KUKA KRL program: EPS_2_251692_SAMH04_A_20251205090700.src

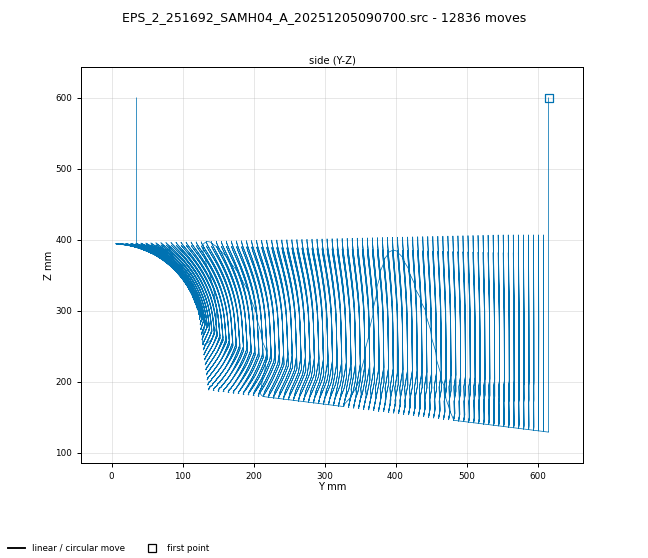
[picture p0: tool path of EPS_2_251692_SAMH04_A_20251205090700.src, 12836 of 12838 moves have a stored position in this frame; points joined in program order, loops and branches not executed]
&ACCESS RVP
&REL 4
&COMMENT QRS 19112012
&PARAM EDITMASK = *
DEF PART()
EXT BAS (BAS_COMMAND :IN,REAL :IN )
INT I
BAS (#INITMOV,0 )

;KUKA QRS Post kuka4.cps  Date:22-06-2017 !

File_ID=2946

QRS_PRE_INIT()

;Init var - Until changes are made in qrs_pre_init
Outlet_Square_prg=0
Inlet_1_Square_prg=0
Inlet_2_Square_prg=0
Inlet_3_Square_prg=0
Inlet_4_Square_prg=0
Inlet_5_Square_prg=0

Outlet_1={X 0.000, Y 546.330, Z 306.500, B 0.000, E1 0.000 }
Inlet_1={X 0.000, Y 548.110, Z 281.500, B 0.000, E1 180.000 }
Outlet_1_type=201
Inlet_1_type=201
;QRS#1=Sidecore dimensions
;QRS#2=200-8" PVC SDR 35
;QRS#3=200-8" PVC SDR 35
;QRS#4=
;QRS#5=
;QRS#6=
;QRS#7=
;QRS#8=
;QRS#9=12-08 PSX
;QRS#10=12-08 PSX
;QRS#11=
;QRS#12=
;QRS#13=
;QRS#14=
;QRS#15=
;QRS#16=1220x127x686 2,25'
;QRS#17=EPS Height
;QRS#18=407
;QRS#19=*
;QRS#20= UPDATED VERSION 22-06-2017
;QRS#21=*
Outlet_Square=0100
Inlet_1_Square=0100
Inlet_2_Square=0
Inlet_3_Square=0
Inlet_4_Square=0
Inlet_5_Square=0
Mill_Square=1
Outlet_Square_Prg=204
Inlet_1_Square_prg=204

QRS_INIT()

$ADVANCE=5

; T1
PTP {E1 173.62,E2 173.62}
PTP {X 0,Y 615.48,A -85,B 0,C 180,E1 173.62,E2 173.62,E3 0,E4 0,E5 0,E6 0}
QRS_SPEED_INIT()
LIN {X 0,Y 615.48,Z 600,A -85,B 0,C 180,E1 173.62,E2 173.62,E3 0,E4 0,E5 0,E6 0} C_VEL
LIN {X 0,Y 615.48,Z 139.368,A -85,B 0,C 180,E1 173.62,E2 173.62} C_VEL
LIN {X 0,Y 615.48,Z 131.192,A -85,B 0,C 180,E1 173.62,E2 173.62} C_VEL
LIN {X 0,Y 615.471,Z 129.192,A -85,B 0,C 180,E1 173.434,E2 173.434} C_VEL
LIN {X 0,Y 615.484,Z 129.195,A -85,B 0,C 180,E1 170.801,E2 170.801} C_VEL
LIN {X 0,Y 615.485,Z 129.184,A -85,B 0,C 180,E1 168.139,E2 168.139} C_VEL
LIN {X 0,Y 615.481,Z 129.196,A -85,B 0,C 180,E1 165.451,E2 165.451} C_VEL
LIN {X 0,Y 615.483,Z 129.188,A -85,B 0,C 180,E1 162.729,E2 162.729} C_VEL
LIN {X 0,Y 615.475,Z 129.189,A -85,B 0,C 180,E1 159.967,E2 159.967} C_VEL
LIN {X 0,Y 615.483,Z 129.194,A -85,B 0,C 180,E1 157.155,E2 157.155} C_VEL
LIN {X 0,Y 615.481,Z 129.186,A -85,B 0,C 180,E1 154.284,E2 154.284} C_VEL
LIN {X 0,Y 615.494,Z 129.199,A -85,B 0,C 180,E1 151.548,E2 151.548} C_VEL
LIN {X 0,Y 615.485,Z 129.185,A -85,B 0,C 180,E1 148.914,E2 148.914} C_VEL
LIN {X 0,Y 615.483,Z 129.186,A -85,B 0,C 180,E1 146.466,E2 146.466} C_VEL
LIN {X 0,Y 615.481,Z 129.195,A -85,B 0,C 180,E1 143.575,E2 143.575} C_VEL
LIN {X 0,Y 615.494,Z 129.181,A -85,B 0,C 180,E1 140.937,E2 140.937} C_VEL
LIN {X 0,Y 615.488,Z 129.199,A -85,B 0,C 180,E1 137.92,E2 137.92} C_VEL
LIN {X 0,Y 615.495,Z 129.182,A -85,B 0,C 180,E1 134.932,E2 134.932} C_VEL
LIN {X 0,Y 615.489,Z 129.198,A -85,B 0,C 180,E1 132.08,E2 132.08} C_VEL
LIN {X 0,Y 615.47,Z 129.192,A -85,B 0,C 180,E1 129.751,E2 129.751} C_VEL
LIN {X 0,Y 615.488,Z 129.186,A -85,B 0,C 180,E1 126.936,E2 126.936} C_VEL
LIN {X 0,Y 615.47,Z 129.194,A -85,B 0,C 180,E1 124.023,E2 124.023} C_VEL
LIN {X 0,Y 615.469,Z 129.188,A -85,B 0,C 180,E1 121.686,E2 121.686} C_VEL
LIN {X 0,Y 615.486,Z 129.184,A -85,B 0,C 180,E1 119.406,E2 119.406} C_VEL
LIN {X 0,Y 615.478,Z 129.197,A -85,B 0,C 180,E1 116.444,E2 116.444} C_VEL
LIN {X 0,Y 615.465,Z 129.189,A -85,B 0,C 180,E1 114.003,E2 114.003} C_VEL
LIN {X 0,Y 615.495,Z 129.184,A -85,B 0,C 180,E1 111.432,E2 111.432} C_VEL
LIN {X 0,Y 615.495,Z 129.385,A -85,B 0,C 180,E1 109.468,E2 109.468} C_VEL
LIN {X 0,Y 615.486,Z 146.128,A -85,B 0,C 180,E1 106.757,E2 106.757} C_VEL
LIN {X 0,Y 615.491,Z 164.181,A -85,B 0,C 180,E1 103.874,E2 103.874} C_VEL
LIN {X 0,Y 615.487,Z 170.814,A -85,B 0,C 180,E1 102.824,E2 102.824} C_VEL
LIN {X 0,Y 615.486,Z 278.794,A -85,B 0,C 180,E1 101.527,E2 101.527} C_VEL
LIN {X 0,Y 615.476,Z 291.742,A -85,B 0,C 180,E1 101.235,E2 101.235} C_VEL
LIN {X 0,Y 615.488,Z 303.661,A -85,B 0,C 180,E1 100.84,E2 100.84} C_VEL
LIN {X 0,Y 615.481,Z 316.197,A -85,B 0,C 180,E1 100.278,E2 100.278} C_VEL
LIN {X 0,Y 615.494,Z 327.576,A -85,B 0,C 180,E1 99.613,E2 99.613} C_VEL
LIN {X 0,Y 615.498,Z 337.823,A -85,B 0,C 180,E1 98.867,E2 98.867} C_VEL
LIN {X 0,Y 615.498,Z 347.034,A -85,B 0,C 180,E1 98.041,E2 98.041} C_VEL
LIN {X 0,Y 615.499,Z 355.892,A -85,B 0,C 180,E1 97.057,E2 97.057} C_VEL
LIN {X 0,Y 615.497,Z 363.123,A -85,B 0,C 180,E1 96.063,E2 96.063} C_VEL
LIN {X 0,Y 615.497,Z 367.958,A -85,B 0,C 180,E1 95.241,E2 95.241} C_VEL
LIN {X 0,Y 615.494,Z 372.658,A -85,B 0,C 180,E1 94.256,E2 94.256} C_VEL
LIN {X 0,Y 615.494,Z 376.254,A -85,B 0,C 180,E1 93.273,E2 93.273} C_VEL
LIN {X 0,Y 615.496,Z 378.115,A -85,B 0,C 180,E1 92.618,E2 92.618} C_VEL
LIN {X 0,Y 615.5,Z 379.533,A -85,B 0,C 180,E1 91.963,E2 91.963} C_VEL
LIN {X 0,Y 615.496,Z 381.141,A -85,B 0,C 180,E1 90.654,E2 90.654} C_VEL
LIN {X 0,Y 615.495,Z 381.384,A -85,B 0,C 180,E1 90,E2 90} C_VEL
LIN {X 0,Y 615.495,Z 381.206,A -85,B 0,C 180,E1 89.346,E2 89.346} C_VEL
LIN {X 0,Y 615.5,Z 379.682,A -85,B 0,C 180,E1 88.037,E2 88.037} C_VEL
LIN {X 0,Y 615.498,Z 378.341,A -85,B 0,C 180,E1 87.382,E2 87.382} C_VEL
LIN {X 0,Y 615.496,Z 375.494,A -85,B 0,C 180,E1 86.399,E2 86.399} C_VEL
LIN {X 0,Y 615.498,Z 371.634,A -85,B 0,C 180,E1 85.416,E2 85.416} C_VEL
LIN {X 0,Y 615.498,Z 366.652,A -85,B 0,C 180,E1 84.43,E2 84.43} C_VEL
LIN {X 0,Y 615.496,Z 360.208,A -85,B 0,C 180,E1 83.418,E2 83.418} C_VEL
LIN {X 0,Y 615.497,Z 352.537,A -85,B 0,C 180,E1 82.455,E2 82.455} C_VEL
LIN {X 0,Y 615.498,Z 342.759,A -85,B 0,C 180,E1 81.464,E2 81.464} C_VEL
LIN {X 0,Y 615.498,Z 332.494,A -85,B 0,C 180,E1 80.636,E2 80.636} C_VEL
LIN {X 0,Y 615.48,Z 320.933,A -85,B 0,C 180,E1 79.889,E2 79.889} C_VEL
LIN {X 0,Y 615.494,Z 309.074,A -85,B 0,C 180,E1 79.293,E2 79.293} C_VEL
LIN {X 0,Y 615.478,Z 296.164,A -85,B 0,C 180,E1 78.807,E2 78.807} C_VEL
LIN {X 0,Y 615.485,Z 283.563,A -85,B 0,C 180,E1 78.473,E2 78.473} C_VEL
LIN {X 0,Y 615.493,Z 270.44,A -85,B 0,C 180,E1 78.265,E2 78.265} C_VEL
LIN {X 0,Y 615.493,Z 170.852,A -85,B 0,C 180,E1 77.093,E2 77.093} C_VEL
LIN {X 0,Y 615.491,Z 152.002,A -85,B 0,C 180,E1 74.095,E2 74.095} C_VEL
LIN {X 0,Y 615.477,Z 134.992,A -85,B 0,C 180,E1 71.354,E2 71.354} C_VEL
LIN {X 0,Y 615.489,Z 129.185,A -85,B 0,C 180,E1 70.402,E2 70.402} C_VEL
LIN {X 0,Y 615.46,Z 129.193,A -85,B 0,C 180,E1 67.661,E2 67.661} C_VEL
LIN {X 0,Y 615.492,Z 129.195,A -85,B 0,C 180,E1 65.009,E2 65.009} C_VEL
LIN {X 0,Y 615.462,Z 129.19,A -85,B 0,C 180,E1 62.084,E2 62.084} C_VEL
LIN {X 0,Y 615.465,Z 129.194,A -85,B 0,C 180,E1 59.839,E2 59.839} C_VEL
LIN {X 0,Y 615.482,Z 129.2,A -85,B 0,C 180,E1 57.542,E2 57.542} C_VEL
LIN {X 0,Y 615.489,Z 129.192,A -85,B 0,C 180,E1 55.185,E2 55.185} C_VEL
LIN {X 0,Y 615.491,Z 129.183,A -85,B 0,C 180,E1 52.758,E2 52.758} C_VEL
LIN {X 0,Y 615.476,Z 129.197,A -85,B 0,C 180,E1 49.913,E2 49.913} C_VEL
LIN {X 0,Y 615.488,Z 129.184,A -85,B 0,C 180,E1 46.953,E2 46.953} C_VEL
LIN {X 0,Y 615.475,Z 129.195,A -85,B 0,C 180,E1 44.151,E2 44.151} C_VEL
LIN {X 0,Y 615.484,Z 129.19,A -85,B 0,C 180,E1 41.474,E2 41.474} C_VEL
LIN {X 0,Y 615.482,Z 129.184,A -85,B 0,C 180,E1 38.905,E2 38.905} C_VEL
LIN {X 0,Y 615.476,Z 129.194,A -85,B 0,C 180,E1 36.426,E2 36.426} C_VEL
LIN {X 0,Y 615.485,Z 129.186,A -85,B 0,C 180,E1 33.534,E2 33.534} C_VEL
LIN {X 0,Y 615.477,Z 129.188,A -85,B 0,C 180,E1 30.921,E2 30.921} C_VEL
LIN {X 0,Y 615.489,Z 129.198,A -85,B 0,C 180,E1 28.451,E2 28.451} C_VEL
LIN {X 0,Y 615.486,Z 129.184,A -85,B 0,C 180,E1 25.569,E2 25.569} C_VEL
LIN {X 0,Y 615.48,Z 129.193,A -85,B 0,C 180,E1 22.845,E2 22.845} C_VEL
LIN {X 0,Y 615.489,Z 129.202,A -85,B 0,C 180,E1 20.558,E2 20.558} C_VEL
LIN {X 0,Y 615.478,Z 129.187,A -85,B 0,C 180,E1 17.957,E2 17.957} C_VEL
LIN {X 0,Y 615.481,Z 129.189,A -85,B 0,C 180,E1 15.226,E2 15.226} C_VEL
LIN {X 0,Y 615.481,Z 129.195,A -85,B 0,C 180,E1 12.53,E2 12.53} C_VEL
LIN {X 0,Y 615.493,Z 129.182,A -85,B 0,C 180,E1 9.862,E2 9.862} C_VEL
LIN {X 0,Y 615.486,Z 129.195,A -85,B 0,C 180,E1 7.216,E2 7.216} C_VEL
LIN {X 0,Y 615.472,Z 129.192,A -85,B 0,C 180,E1 4.585,E2 4.585} C_VEL
LIN {X 0,Y 615.5,Z 129.181,A -85,B 0,C 180,E1 1.963,E2 1.963} C_VEL
LIN {X 0,Y 615.492,Z 129.197,A -85,B 0,C 180,E1 -0.654,E2 -0.654} C_VEL
LIN {X 0,Y 615.468,Z 129.191,A -85,B 0,C 180,E1 -3.273,E2 -3.273} C_VEL
LIN {X 0,Y 615.498,Z 129.182,A -85,B 0,C 180,E1 -5.898,E2 -5.898} C_VEL
LIN {X 0,Y 615.49,Z 129.202,A -85,B 0,C 180,E1 -8.537,E2 -8.537} C_VEL
LIN {X 0,Y 615.465,Z 129.19,A -85,B 0,C 180,E1 -11.194,E2 -11.194} C_VEL
LIN {X 0,Y 615.49,Z 129.188,A -85,B 0,C 180,E1 -13.935,E2 -13.935} C_VEL
LIN {X 0,Y 615.475,Z 129.196,A -85,B 0,C 180,E1 -16.587,E2 -16.587} C_VEL
LIN {X 0,Y 615.477,Z 129.186,A -85,B 0,C 180,E1 -19.338,E2 -19.338} C_VEL
LIN {X 0,Y 615.477,Z 129.198,A -85,B 0,C 180,E1 -22.344,E2 -22.344} C_VEL
LIN {X 0,Y 615.461,Z 129.189,A -85,B 0,C 180,E1 -24.993,E2 -24.993} C_VEL
LIN {X 0,Y 615.487,Z 129.201,A -85,B 0,C 180,E1 -27.915,E2 -27.915} C_VEL
LIN {X 0,Y 615.473,Z 129.197,A -85,B 0,C 180,E1 -30.161,E2 -30.161} C_VEL
LIN {X 0,Y 615.454,Z 129.193,A -85,B 0,C 180,E1 -32.46,E2 -32.46} C_VEL
LIN {X 0,Y 615.462,Z 129.189,A -85,B 0,C 180,E1 -34.817,E2 -34.817} C_VEL
LIN {X 0,Y 615.496,Z 129.187,A -85,B 0,C 180,E1 -37.242,E2 -37.242} C_VEL
LIN {X 0,Y 615.453,Z 129.196,A -85,B 0,C 180,E1 -40.085,E2 -40.085} C_VEL
LIN {X 0,Y 615.448,Z 129.192,A -85,B 0,C 180,E1 -42.357,E2 -42.357} C_VEL
LIN {X 0,Y 615.497,Z 129.189,A -85,B 0,C 180,E1 -45.068,E2 -45.068} C_VEL
LIN {X 0,Y 615.449,Z 129.195,A -85,B 0,C 180,E1 -47.924,E2 -47.924} C_VEL
LIN {X 0,Y 615.444,Z 129.193,A -85,B 0,C 180,E1 -50.247,E2 -50.247} C_VEL
LIN {X 0,Y 615.49,Z 129.197,A -85,B 0,C 180,E1 -53.063,E2 -53.063} C_VEL
LIN {X 0,Y 615.44,Z 129.194,A -85,B 0,C 180,E1 -55.975,E2 -55.975} C_VEL
LIN {X 0,Y 615.488,Z 129.199,A -85,B 0,C 180,E1 -58.914,E2 -58.914} C_VEL
LIN {X 0,Y 615.441,Z 129.196,A -85,B 0,C 180,E1 -61.558,E2 -61.558} C_VEL
LIN {X 0,Y 615.438,Z 129.196,A -85,B 0,C 180,E1 -63.554,E2 -63.554} C_VEL
LIN {X 0,Y 615.444,Z 129.194,A -85,B 0,C 180,E1 -66.001,E2 -66.001} C_VEL
LIN {X 0,Y 615.449,Z 129.225,A -85,B 0,C 180,E1 -68.039,E2 -68.039} C_VEL
LIN {X 0,Y 615.481,Z 149.073,A -85,B 0,C 180,E1 -70.835,E2 -70.835} C_VEL
LIN {X 0,Y 615.46,Z 167.661,A -85,B 0,C 180,E1 -73.413,E2 -73.413} C_VEL
LIN {X 0,Y 615.483,Z 187.465,A -85,B 0,C 180,E1 -76.126,E2 -76.126} C_VEL
LIN {X 0,Y 615.462,Z 195.117,A -85,B 0,C 180,E1 -77.134,E2 -77.134} C_VEL
LIN {X 0,Y 615.488,Z 302.834,A -85,B 0,C 180,E1 -78.411,E2 -78.411} C_VEL
LIN {X 0,Y 615.477,Z 315.348,A -85,B 0,C 180,E1 -78.682,E2 -78.682} C_VEL
LIN {X 0,Y 615.488,Z 328.617,A -85,B 0,C 180,E1 -79.113,E2 -79.113} C_VEL
LIN {X 0,Y 615.477,Z 340.48,A -85,B 0,C 180,E1 -79.639,E2 -79.639} C_VEL
LIN {X 0,Y 615.494,Z 351.995,A -85,B 0,C 180,E1 -80.304,E2 -80.304} C_VEL
LIN {X 0,Y 615.499,Z 362.342,A -85,B 0,C 180,E1 -81.05,E2 -81.05} C_VEL
LIN {X 0,Y 615.497,Z 370.812,A -85,B 0,C 180,E1 -81.794,E2 -81.794} C_VEL
LIN {X 0,Y 615.498,Z 378.607,A -85,B 0,C 180,E1 -82.62,E2 -82.62} C_VEL
LIN {X 0,Y 615.496,Z 386.203,A -85,B 0,C 180,E1 -83.608,E2 -83.608} C_VEL
LIN {X 0,Y 615.498,Z 393.205,A -85,B 0,C 180,E1 -84.759,E2 -84.759} C_VEL
LIN {X 0,Y 615.494,Z 397.852,A -85,B 0,C 180,E1 -85.744,E2 -85.744} C_VEL
LIN {X 0,Y 615.494,Z 401.399,A -85,B 0,C 180,E1 -86.727,E2 -86.727} C_VEL
LIN {X 0,Y 615.497,Z 403.233,A -85,B 0,C 180,E1 -87.382,E2 -87.382} C_VEL
LIN {X 0,Y 615.5,Z 404.607,A -85,B 0,C 180,E1 -88.037,E2 -88.037} C_VEL
LIN {X 0,Y 615.496,Z 406.173,A -85,B 0,C 180,E1 -89.346,E2 -89.346} C_VEL
LIN {X 0,Y 615.494,Z 406.389,A -85,B 0,C 180,E1 -90,E2 -90} C_VEL
LIN {X 0,Y 615.495,Z 405.58,A -85,B 0,C 180,E1 -91.309,E2 -91.309} C_VEL
LIN {X 0,Y 615.5,Z 404.607,A -85,B 0,C 180,E1 -91.963,E2 -91.963} C_VEL
LIN {X 0,Y 615.497,Z 403.233,A -85,B 0,C 180,E1 -92.618,E2 -92.618} C_VEL
LIN {X 0,Y 615.496,Z 400.349,A -85,B 0,C 180,E1 -93.601,E2 -93.601} C_VEL
LIN {X 0,Y 615.498,Z 396.441,A -85,B 0,C 180,E1 -94.584,E2 -94.584} C_VEL
LIN {X 0,Y 615.499,Z 391.405,A -85,B 0,C 180,E1 -95.57,E2 -95.57} C_VEL
LIN {X 0,Y 615.497,Z 384.869,A -85,B 0,C 180,E1 -96.583,E2 -96.583} C_VEL
LIN {X 0,Y 615.497,Z 377.133,A -85,B 0,C 180,E1 -97.545,E2 -97.545} C_VEL
LIN {X 0,Y 615.498,Z 369.045,A -85,B 0,C 180,E1 -98.371,E2 -98.371} C_VEL
LIN {X 0,Y 615.499,Z 359.167,A -85,B 0,C 180,E1 -99.199,E2 -99.199} C_VEL
LIN {X 0,Y 615.488,Z 347.982,A -85,B 0,C 180,E1 -99.945,E2 -99.945} C_VEL
LIN {X 0,Y 615.482,Z 337.023,A -85,B 0,C 180,E1 -100.527,E2 -100.527} C_VEL
LIN {X 0,Y 615.48,Z 324.49,A -85,B 0,C 180,E1 -101.04,E2 -101.04} C_VEL
LIN {X 0,Y 615.479,Z 312.067,A -85,B 0,C 180,E1 -101.402,E2 -101.402} C_VEL
LIN {X 0,Y 615.493,Z 298.465,A -85,B 0,C 180,E1 -101.652,E2 -101.652} C_VEL
LIN {X 0,Y 615.463,Z 194.734,A -85,B 0,C 180,E1 -102.887,E2 -102.887} C_VEL
LIN {X 0,Y 615.498,Z 173.851,A -85,B 0,C 180,E1 -105.735,E2 -105.735} C_VEL
LIN {X 0,Y 615.49,Z 153.088,A -85,B 0,C 180,E1 -108.605,E2 -108.605} C_VEL
LIN {X 0,Y 615.498,Z 132.948,A -85,B 0,C 180,E1 -111.431,E2 -111.431} C_VEL
LIN {X 0,Y 615.447,Z 129.194,A -85,B 0,C 180,E1 -111.983,E2 -111.983} C_VEL
LIN {X 0,Y 615.434,Z 129.195,A -85,B 0,C 180,E1 -114.274,E2 -114.274} C_VEL
LIN {X 0,Y 615.491,Z 129.2,A -85,B 0,C 180,E1 -117.045,E2 -117.045} C_VEL
LIN {X 0,Y 615.451,Z 129.192,A -85,B 0,C 180,E1 -119.788,E2 -119.788} C_VEL
LIN {X 0,Y 615.439,Z 129.197,A -85,B 0,C 180,E1 -122.323,E2 -122.323} C_VEL
LIN {X 0,Y 615.49,Z 129.2,A -85,B 0,C 180,E1 -124.815,E2 -124.815} C_VEL
LIN {X 0,Y 615.488,Z 129.189,A -85,B 0,C 180,E1 -127.242,E2 -127.242} C_VEL
LIN {X 0,Y 615.443,Z 129.193,A -85,B 0,C 180,E1 -129.753,E2 -129.753} C_VEL
LIN {X 0,Y 615.466,Z 129.198,A -85,B 0,C 180,E1 -132.355,E2 -132.355} C_VEL
LIN {X 0,Y 615.491,Z 129.187,A -85,B 0,C 180,E1 -135.068,E2 -135.068} C_VEL
LIN {X 0,Y 615.447,Z 129.193,A -85,B 0,C 180,E1 -137.643,E2 -137.643} C_VEL
LIN {X 0,Y 615.48,Z 129.199,A -85,B 0,C 180,E1 -140.249,E2 -140.249} C_VEL
LIN {X 0,Y 615.473,Z 129.188,A -85,B 0,C 180,E1 -143.065,E2 -143.065} C_VEL
LIN {X 0,Y 615.455,Z 129.19,A -85,B 0,C 180,E1 -145.304,E2 -145.304} C_VEL
LIN {X 0,Y 615.456,Z 129.195,A -85,B 0,C 180,E1 -147.674,E2 -147.674} C_VEL
LIN {X 0,Y 615.497,Z 129.198,A -85,B 0,C 180,E1 -150.204,E2 -150.204} C_VEL
LIN {X 0,Y 615.464,Z 129.188,A -85,B 0,C 180,E1 -152.959,E2 -152.959} C_VEL
LIN {X 0,Y 615.461,Z 129.189,A -85,B 0,C 180,E1 -155.007,E2 -155.007} C_VEL
LIN {X 0,Y 615.473,Z 129.198,A -85,B 0,C 180,E1 -157.657,E2 -157.657} C_VEL
LIN {X 0,Y 615.477,Z 129.186,A -85,B 0,C 180,E1 -160.662,E2 -160.662} C_VEL
LIN {X 0,Y 615.467,Z 129.197,A -85,B 0,C 180,E1 -163.413,E2 -163.413} C_VEL
LIN {X 0,Y 615.492,Z 129.187,A -85,B 0,C 180,E1 -166.126,E2 -166.126} C_VEL
LIN {X 0,Y 615.462,Z 129.19,A -85,B 0,C 180,E1 -168.806,E2 -168.806} C_VEL
LIN {X 0,Y 615.488,Z 129.202,A -85,B 0,C 180,E1 -171.463,E2 -171.463} C_VEL
LIN {X 0,Y 615.498,Z 129.182,A -85,B 0,C 180,E1 -174.102,E2 -174.102} C_VEL
LIN {X 0,Y 615.465,Z 129.191,A -85,B 0,C 180,E1 -176.727,E2 -176.727} C_VEL
LIN {X 0,Y 615.494,Z 129.198,A -85,B 0,C 180,E1 -179.346,E2 -179.346} C_VEL
LIN {X 0,Y 615.5,Z 129.181,A -85,B 0,C 180,E1 -181.963,E2 -181.963} C_VEL
LIN {X 0,Y 615.469,Z 129.192,A -85,B 0,C 180,E1 -184.585,E2 -184.585} C_VEL
LIN {X 0,Y 615.471,Z 129.192,A -85,B 0,C 180,E1 -186.566,E2 -186.566} C_VEL
LIN {X 0,Y 614.806,Z 129.344,A -85,B 0,C 180,E1 -187.112,E2 -187.112} C_VEL
LIN {X 0,Y 611.978,Z 129.748,A -85,B 0,C 180,E1 -187.998,E2 -187.998} C_VEL
LIN {X 0,Y 609.585,Z 130.062,A -85,B 0,C 180,E1 -188.711,E2 -188.711} C_VEL
LIN {X 0,Y 608.549,Z 130.181,A -85,B 0,C 180,E1 -189.26,E2 -189.26} C_VEL
LIN {X 0,Y 608.46,Z 130.189,A -85,B 0,C 180,E1 -189.446,E2 -189.446} C_VEL
LIN {X 0,Y 608.459,Z 130.187,A -85,B 0,C 180,E1 -192,E2 -192} C_VEL
LIN {X 0,Y 608.471,Z 130.195,A -85,B 0,C 180,E1 -194.721,E2 -194.721} C_VEL
LIN {X 0,Y 608.448,Z 130.189,A -85,B 0,C 180,E1 -197.477,E2 -197.477} C_VEL
LIN {X 0,Y 608.457,Z 130.192,A -85,B 0,C 180,E1 -200.274,E2 -200.274} C_VEL
LIN {X 0,Y 608.459,Z 130.196,A -85,B 0,C 180,E1 -202.477,E2 -202.477} C_VEL
LIN {X 0,Y 608.449,Z 130.188,A -85,B 0,C 180,E1 -205.301,E2 -205.301} C_VEL
LIN {X 0,Y 608.446,Z 130.189,A -85,B 0,C 180,E1 -207.518,E2 -207.518} C_VEL
LIN {X 0,Y 608.463,Z 130.191,A -85,B 0,C 180,E1 -209.971,E2 -209.971} C_VEL
LIN {X 0,Y 608.458,Z 130.188,A -85,B 0,C 180,E1 -212.88,E2 -212.88} C_VEL
LIN {X 0,Y 608.437,Z 130.19,A -85,B 0,C 180,E1 -215.278,E2 -215.278} C_VEL
LIN {X 0,Y 608.472,Z 130.19,A -85,B 0,C 180,E1 -217.746,E2 -217.746} C_VEL
LIN {X 0,Y 608.451,Z 130.193,A -85,B 0,C 180,E1 -220.329,E2 -220.329} C_VEL
LIN {X 0,Y 608.453,Z 130.188,A -85,B 0,C 180,E1 -222.96,E2 -222.96} C_VEL
LIN {X 0,Y 608.463,Z 130.195,A -85,B 0,C 180,E1 -225.736,E2 -225.736} C_VEL
LIN {X 0,Y 608.456,Z 130.187,A -85,B 0,C 180,E1 -228.659,E2 -228.659} C_VEL
LIN {X 0,Y 608.463,Z 130.196,A -85,B 0,C 180,E1 -231.761,E2 -231.761} C_VEL
LIN {X 0,Y 608.444,Z 130.194,A -85,B 0,C 180,E1 -233.955,E2 -233.955} C_VEL
LIN {X 0,Y 608.444,Z 130.189,A -85,B 0,C 180,E1 -236.328,E2 -236.328} C_VEL
LIN {X 0,Y 608.449,Z 130.189,A -85,B 0,C 180,E1 -238.733,E2 -238.733} C_VEL
LIN {X 0,Y 608.473,Z 130.196,A -85,B 0,C 180,E1 -241.381,E2 -241.381} C_VEL
LIN {X 0,Y 608.436,Z 130.191,A -85,B 0,C 180,E1 -243.964,E2 -243.964} C_VEL
LIN {X 0,Y 608.453,Z 130.192,A -85,B 0,C 180,E1 -246.876,E2 -246.876} C_VEL
LIN {X 0,Y 608.462,Z 130.195,A -85,B 0,C 180,E1 -249.324,E2 -249.324} C_VEL
LIN {X 0,Y 608.485,Z 130.23,A -85,B 0,C 180,E1 -250.431,E2 -250.431} C_VEL
LIN {X 0,Y 608.499,Z 146.216,A -85,B 0,C 180,E1 -253.044,E2 -253.044} C_VEL
LIN {X 0,Y 608.474,Z 163.27,A -85,B 0,C 180,E1 -255.792,E2 -255.792} C_VEL
LIN {X 0,Y 608.459,Z 171.064,A -85,B 0,C 180,E1 -257.036,E2 -257.036} C_VEL
LIN {X 0,Y 608.556,Z 277.795,A -85,B 0,C 180,E1 -258.319,E2 -258.319} C_VEL
LIN {X 0,Y 608.525,Z 291.115,A -85,B 0,C 180,E1 -258.614,E2 -258.614} C_VEL
LIN {X 0,Y 608.508,Z 303.627,A -85,B 0,C 180,E1 -259.027,E2 -259.027} C_VEL
LIN {X 0,Y 608.504,Z 314.736,A -85,B 0,C 180,E1 -259.519,E2 -259.519} C_VEL
LIN {X 0,Y 608.484,Z 326.513,A -85,B 0,C 180,E1 -260.191,E2 -260.191} C_VEL
LIN {X 0,Y 608.485,Z 337.025,A -85,B 0,C 180,E1 -260.946,E2 -260.946} C_VEL
LIN {X 0,Y 608.475,Z 345.634,A -85,B 0,C 180,E1 -261.699,E2 -261.699} C_VEL
LIN {X 0,Y 608.47,Z 353.564,A -85,B 0,C 180,E1 -262.534,E2 -262.534} C_VEL
LIN {X 0,Y 608.468,Z 361.07,A -85,B 0,C 180,E1 -263.497,E2 -263.497} C_VEL
LIN {X 0,Y 608.451,Z 366.609,A -85,B 0,C 180,E1 -264.366,E2 -264.366} C_VEL
LIN {X 0,Y 608.431,Z 371.751,A -85,B 0,C 180,E1 -265.362,E2 -265.362} C_VEL
LIN {X 0,Y 608.449,Z 375.741,A -85,B 0,C 180,E1 -266.358,E2 -266.358} C_VEL
LIN {X 0,Y 608.425,Z 378.691,A -85,B 0,C 180,E1 -267.352,E2 -267.352} C_VEL
LIN {X 0,Y 608.445,Z 380.127,A -85,B 0,C 180,E1 -268.014,E2 -268.014} C_VEL
LIN {X 0,Y 608.439,Z 381.752,A -85,B 0,C 180,E1 -269.338,E2 -269.338} C_VEL
LIN {X 0,Y 608.435,Z 381.995,A -85,B 0,C 180,E1 -270,E2 -270} C_VEL
LIN {X 0,Y 608.438,Z 381.815,A -85,B 0,C 180,E1 -270.662,E2 -270.662} C_VEL
LIN {X 0,Y 608.445,Z 380.276,A -85,B 0,C 180,E1 -271.986,E2 -271.986} C_VEL
LIN {X 0,Y 608.426,Z 378.918,A -85,B 0,C 180,E1 -272.648,E2 -272.648} C_VEL
LIN {X 0,Y 608.449,Z 376.042,A -85,B 0,C 180,E1 -273.642,E2 -273.642} C_VEL
LIN {X 0,Y 608.433,Z 372.143,A -85,B 0,C 180,E1 -274.638,E2 -274.638} C_VEL
LIN {X 0,Y 608.45,Z 367.112,A -85,B 0,C 180,E1 -275.634,E2 -275.634} C_VEL
LIN {X 0,Y 608.441,Z 360.795,A -85,B 0,C 180,E1 -276.633,E2 -276.633} C_VEL
LIN {X 0,Y 608.475,Z 352.879,A -85,B 0,C 180,E1 -277.633,E2 -277.633} C_VEL
LIN {X 0,Y 608.472,Z 343.037,A -85,B 0,C 180,E1 -278.636,E2 -278.636} C_VEL
LIN {X 0,Y 608.48,Z 332.715,A -85,B 0,C 180,E1 -279.473,E2 -279.473} C_VEL
LIN {X 0,Y 608.476,Z 321.101,A -85,B 0,C 180,E1 -280.229,E2 -280.229} C_VEL
LIN {X 0,Y 608.518,Z 308.898,A -85,B 0,C 180,E1 -280.844,E2 -280.844} C_VEL
LIN {X 0,Y 608.52,Z 296.264,A -85,B 0,C 180,E1 -281.323,E2 -281.323} C_VEL
LIN {X 0,Y 608.544,Z 283.648,A -85,B 0,C 180,E1 -281.66,E2 -281.66} C_VEL
LIN {X 0,Y 608.556,Z 270.548,A -85,B 0,C 180,E1 -281.871,E2 -281.871} C_VEL
LIN {X 0,Y 608.462,Z 171.029,A -85,B 0,C 180,E1 -283.059,E2 -283.059} C_VEL
LIN {X 0,Y 608.496,Z 153.169,A -85,B 0,C 180,E1 -285.921,E2 -285.921} C_VEL
LIN {X 0,Y 608.496,Z 135.934,A -85,B 0,C 180,E1 -288.722,E2 -288.722} C_VEL
LIN {X 0,Y 608.452,Z 130.189,A -85,B 0,C 180,E1 -289.702,E2 -289.702} C_VEL
LIN {X 0,Y 608.447,Z 130.192,A -85,B 0,C 180,E1 -292.473,E2 -292.473} C_VEL
LIN {X 0,Y 608.453,Z 130.19,A -85,B 0,C 180,E1 -295.301,E2 -295.301} C_VEL
LIN {X 0,Y 608.442,Z 130.189,A -85,B 0,C 180,E1 -297.518,E2 -297.518} C_VEL
LIN {X 0,Y 608.449,Z 130.189,A -85,B 0,C 180,E1 -299.968,E2 -299.968} C_VEL
LIN {X 0,Y 608.458,Z 130.192,A -85,B 0,C 180,E1 -302.879,E2 -302.879} C_VEL
LIN {X 0,Y 608.435,Z 130.19,A -85,B 0,C 180,E1 -305.278,E2 -305.278} C_VEL
LIN {X 0,Y 608.461,Z 130.188,A -85,B 0,C 180,E1 -307.747,E2 -307.747} C_VEL
LIN {X 0,Y 608.447,Z 130.199,A -85,B 0,C 180,E1 -310.328,E2 -310.328} C_VEL
LIN {X 0,Y 608.456,Z 130.188,A -85,B 0,C 180,E1 -312.959,E2 -312.959} C_VEL
LIN {X 0,Y 608.448,Z 130.192,A -85,B 0,C 180,E1 -315.737,E2 -315.737} C_VEL
LIN {X 0,Y 608.462,Z 130.188,A -85,B 0,C 180,E1 -318.658,E2 -318.658} C_VEL
LIN {X 0,Y 608.466,Z 130.188,A -85,B 0,C 180,E1 -321.412,E2 -321.412} C_VEL
LIN {X 0,Y 608.446,Z 130.198,A -85,B 0,C 180,E1 -323.954,E2 -323.954} C_VEL
LIN {X 0,Y 608.464,Z 130.189,A -85,B 0,C 180,E1 -326.329,E2 -326.329} C_VEL
LIN {X 0,Y 608.446,Z 130.188,A -85,B 0,C 180,E1 -328.732,E2 -328.732} C_VEL
LIN {X 0,Y 608.471,Z 130.191,A -85,B 0,C 180,E1 -331.38,E2 -331.38} C_VEL
LIN {X 0,Y 608.47,Z 130.187,A -85,B 0,C 180,E1 -334.279,E2 -334.279} C_VEL
LIN {X 0,Y 608.447,Z 130.19,A -85,B 0,C 180,E1 -336.876,E2 -336.876} C_VEL
LIN {X 0,Y 608.468,Z 130.194,A -85,B 0,C 180,E1 -339.321,E2 -339.321} C_VEL
LIN {X 0,Y 608.446,Z 130.192,A -85,B 0,C 180,E1 -341.828,E2 -341.828} C_VEL
LIN {X 0,Y 608.466,Z 130.187,A -85,B 0,C 180,E1 -344.594,E2 -344.594} C_VEL
LIN {X 0,Y 608.47,Z 130.194,A -85,B 0,C 180,E1 -347.323,E2 -347.323} C_VEL
LIN {X 0,Y 608.46,Z 130.187,A -85,B 0,C 180,E1 -350.023,E2 -350.023} C_VEL
LIN {X 0,Y 608.464,Z 130.191,A -85,B 0,C 180,E1 -352.701,E2 -352.701} C_VEL
LIN {X 0,Y 608.463,Z 130.192,A -85,B 0,C 180,E1 -354.698,E2 -354.698} C_VEL
LIN {X 0,Y 608.464,Z 130.189,A -85,B 0,C 180,E1 -357.352,E2 -357.352} C_VEL
LIN {X 0,Y 608.477,Z 130.185,A -85,B 0,C 180,E1 -360,E2 -360} C_VEL
LIN {X 0,Y 608.478,Z 130.193,A -85,B 0,C 180,E1 -362.648,E2 -362.648} C_VEL
LIN {X 0,Y 608.449,Z 130.189,A -85,B 0,C 180,E1 -365.302,E2 -365.302} C_VEL
LIN {X 0,Y 608.479,Z 130.186,A -85,B 0,C 180,E1 -367.967,E2 -367.967} C_VEL
LIN {X 0,Y 608.46,Z 130.19,A -85,B 0,C 180,E1 -370.952,E2 -370.952} C_VEL
LIN {X 0,Y 608.45,Z 130.188,A -85,B 0,C 180,E1 -373.357,E2 -373.357} C_VEL
LIN {X 0,Y 608.463,Z 130.193,A -85,B 0,C 180,E1 -376.094,E2 -376.094} C_VEL
LIN {X 0,Y 608.445,Z 130.19,A -85,B 0,C 180,E1 -378.87,E2 -378.87} C_VEL
LIN {X 0,Y 608.473,Z 130.188,A -85,B 0,C 180,E1 -381.691,E2 -381.691} C_VEL
LIN {X 0,Y 608.439,Z 130.192,A -85,B 0,C 180,E1 -384.572,E2 -384.572} C_VEL
LIN {X 0,Y 608.468,Z 130.186,A -85,B 0,C 180,E1 -387.206,E2 -387.206} C_VEL
LIN {X 0,Y 608.469,Z 130.195,A -85,B 0,C 180,E1 -389.972,E2 -389.972} C_VEL
LIN {X 0,Y 608.446,Z 130.189,A -85,B 0,C 180,E1 -392.88,E2 -392.88} C_VEL
LIN {X 0,Y 608.439,Z 130.192,A -85,B 0,C 180,E1 -395.278,E2 -395.278} C_VEL
LIN {X 0,Y 608.458,Z 130.196,A -85,B 0,C 180,E1 -397.747,E2 -397.747} C_VEL
LIN {X 0,Y 608.432,Z 130.191,A -85,B 0,C 180,E1 -400.327,E2 -400.327} C_VEL
LIN {X 0,Y 608.45,Z 130.19,A -85,B 0,C 180,E1 -402.96,E2 -402.96} C_VEL
LIN {X 0,Y 608.434,Z 130.195,A -85,B 0,C 180,E1 -405.739,E2 -405.739} C_VEL
LIN {X 0,Y 608.432,Z 130.192,A -85,B 0,C 180,E1 -407.936,E2 -407.936} C_VEL
LIN {X 0,Y 608.441,Z 130.191,A -85,B 0,C 180,E1 -410.706,E2 -410.706} C_VEL
LIN {X 0,Y 608.459,Z 130.195,A -85,B 0,C 180,E1 -413.085,E2 -413.085} C_VEL
LIN {X 0,Y 608.452,Z 130.191,A -85,B 0,C 180,E1 -415.53,E2 -415.53} C_VEL
LIN {X 0,Y 608.429,Z 130.191,A -85,B 0,C 180,E1 -417.904,E2 -417.904} C_VEL
LIN {X 0,Y 608.437,Z 130.19,A -85,B 0,C 180,E1 -420.219,E2 -420.219} C_VEL
LIN {X 0,Y 608.486,Z 130.192,A -85,B 0,C 180,E1 -422.792,E2 -422.792} C_VEL
LIN {X 0,Y 608.425,Z 130.193,A -85,B 0,C 180,E1 -425.428,E2 -425.428} C_VEL
LIN {X 0,Y 608.444,Z 130.313,A -85,B 0,C 180,E1 -427.929,E2 -427.929} C_VEL
LIN {X 0,Y 608.552,Z 145.37,A -85,B 0,C 180,E1 -430.081,E2 -430.081} C_VEL
LIN {X 0,Y 608.485,Z 165.238,A -85,B 0,C 180,E1 -432.871,E2 -432.871} C_VEL
LIN {X 0,Y 608.48,Z 185.106,A -85,B 0,C 180,E1 -435.622,E2 -435.622} C_VEL
LIN {X 0,Y 608.47,Z 195.149,A -85,B 0,C 180,E1 -436.984,E2 -436.984} C_VEL
LIN {X 0,Y 608.547,Z 302.951,A -85,B 0,C 180,E1 -438.277,E2 -438.277} C_VEL
LIN {X 0,Y 608.512,Z 316.219,A -85,B 0,C 180,E1 -438.572,E2 -438.572} C_VEL
LIN {X 0,Y 608.513,Z 328.153,A -85,B 0,C 180,E1 -438.964,E2 -438.964} C_VEL
LIN {X 0,Y 608.499,Z 340.636,A -85,B 0,C 180,E1 -439.519,E2 -439.519} C_VEL
LIN {X 0,Y 608.484,Z 352.198,A -85,B 0,C 180,E1 -440.191,E2 -440.191} C_VEL
LIN {X 0,Y 608.485,Z 362.595,A -85,B 0,C 180,E1 -440.946,E2 -440.946} C_VEL
LIN {X 0,Y 608.475,Z 371.112,A -85,B 0,C 180,E1 -441.699,E2 -441.699} C_VEL
LIN {X 0,Y 608.471,Z 378.961,A -85,B 0,C 180,E1 -442.534,E2 -442.534} C_VEL
LIN {X 0,Y 608.461,Z 386.287,A -85,B 0,C 180,E1 -443.485,E2 -443.485} C_VEL
LIN {X 0,Y 608.451,Z 391.866,A -85,B 0,C 180,E1 -444.366,E2 -444.366} C_VEL
LIN {X 0,Y 608.432,Z 396.95,A -85,B 0,C 180,E1 -445.362,E2 -445.362} C_VEL
LIN {X 0,Y 608.449,Z 400.896,A -85,B 0,C 180,E1 -446.358,E2 -446.358} C_VEL
LIN {X 0,Y 608.425,Z 403.809,A -85,B 0,C 180,E1 -447.352,E2 -447.352} C_VEL
LIN {X 0,Y 608.445,Z 405.201,A -85,B 0,C 180,E1 -448.014,E2 -448.014} C_VEL
LIN {X 0,Y 608.438,Z 406.783,A -85,B 0,C 180,E1 -449.338,E2 -449.338} C_VEL
LIN {X 0,Y 608.434,Z 407,A -85,B 0,C 180,E1 -450,E2 -450} C_VEL
LIN {X 0,Y 608.448,Z 406.184,A -85,B 0,C 180,E1 -451.324,E2 -451.324} C_VEL
LIN {X 0,Y 608.445,Z 405.201,A -85,B 0,C 180,E1 -451.986,E2 -451.986} C_VEL
LIN {X 0,Y 608.425,Z 403.809,A -85,B 0,C 180,E1 -452.648,E2 -452.648} C_VEL
LIN {X 0,Y 608.449,Z 400.896,A -85,B 0,C 180,E1 -453.642,E2 -453.642} C_VEL
LIN {X 0,Y 608.432,Z 396.95,A -85,B 0,C 180,E1 -454.638,E2 -454.638} C_VEL
LIN {X 0,Y 608.438,Z 390.877,A -85,B 0,C 180,E1 -455.801,E2 -455.801} C_VEL
LIN {X 0,Y 608.462,Z 384.235,A -85,B 0,C 180,E1 -456.799,E2 -456.799} C_VEL
LIN {X 0,Y 608.456,Z 375.989,A -85,B 0,C 180,E1 -457.8,E2 -457.8} C_VEL
LIN {X 0,Y 608.472,Z 367.536,A -85,B 0,C 180,E1 -458.636,E2 -458.636} C_VEL
LIN {X 0,Y 608.479,Z 357.091,A -85,B 0,C 180,E1 -459.473,E2 -459.473} C_VEL
LIN {X 0,Y 608.489,Z 346.756,A -85,B 0,C 180,E1 -460.145,E2 -460.145} C_VEL
LIN {X 0,Y 608.519,Z 335.267,A -85,B 0,C 180,E1 -460.74,E2 -460.74} C_VEL
LIN {X 0,Y 608.528,Z 322.891,A -85,B 0,C 180,E1 -461.225,E2 -461.225} C_VEL
LIN {X 0,Y 608.544,Z 309.439,A -85,B 0,C 180,E1 -461.597,E2 -461.597} C_VEL
LIN {X 0,Y 608.554,Z 297.085,A -85,B 0,C 180,E1 -461.808,E2 -461.808} C_VEL
LIN {X 0,Y 608.47,Z 195.144,A -85,B 0,C 180,E1 -463.016,E2 -463.016} C_VEL
LIN {X 0,Y 608.505,Z 175.171,A -85,B 0,C 180,E1 -465.749,E2 -465.749} C_VEL
LIN {X 0,Y 608.509,Z 155.451,A -85,B 0,C 180,E1 -468.498,E2 -468.498} C_VEL
LIN {X 0,Y 608.562,Z 136.677,A -85,B 0,C 180,E1 -471.155,E2 -471.155} C_VEL
LIN {X 0,Y 608.412,Z 130.195,A -85,B 0,C 180,E1 -472.095,E2 -472.095} C_VEL
LIN {X 0,Y 608.425,Z 130.193,A -85,B 0,C 180,E1 -474.572,E2 -474.572} C_VEL
LIN {X 0,Y 608.486,Z 130.192,A -85,B 0,C 180,E1 -477.208,E2 -477.208} C_VEL
LIN {X 0,Y 608.415,Z 130.192,A -85,B 0,C 180,E1 -479.962,E2 -479.962} C_VEL
LIN {X 0,Y 608.428,Z 130.194,A -85,B 0,C 180,E1 -482.517,E2 -482.517} C_VEL
LIN {X 0,Y 608.428,Z 130.194,A -85,B 0,C 180,E1 -485.279,E2 -485.279} C_VEL
LIN {X 0,Y 608.442,Z 130.189,A -85,B 0,C 180,E1 -487.748,E2 -487.748} C_VEL
LIN {X 0,Y 608.433,Z 130.194,A -85,B 0,C 180,E1 -490.327,E2 -490.327} C_VEL
LIN {X 0,Y 608.463,Z 130.187,A -85,B 0,C 180,E1 -493.308,E2 -493.308} C_VEL
LIN {X 0,Y 608.445,Z 130.192,A -85,B 0,C 180,E1 -496.128,E2 -496.128} C_VEL
LIN {X 0,Y 608.459,Z 130.191,A -85,B 0,C 180,E1 -498.824,E2 -498.824} C_VEL
LIN {X 0,Y 608.424,Z 130.191,A -85,B 0,C 180,E1 -501.408,E2 -501.408} C_VEL
LIN {X 0,Y 608.442,Z 130.194,A -85,B 0,C 180,E1 -503.955,E2 -503.955} C_VEL
LIN {X 0,Y 608.464,Z 130.195,A -85,B 0,C 180,E1 -506.329,E2 -506.329} C_VEL
LIN {X 0,Y 608.445,Z 130.191,A -85,B 0,C 180,E1 -508.732,E2 -508.732} C_VEL
LIN {X 0,Y 608.447,Z 130.189,A -85,B 0,C 180,E1 -511.384,E2 -511.384} C_VEL
LIN {X 0,Y 608.438,Z 130.199,A -85,B 0,C 180,E1 -513.964,E2 -513.964} C_VEL
LIN {X 0,Y 608.475,Z 130.192,A -85,B 0,C 180,E1 -516.155,E2 -516.155} C_VEL
LIN {X 0,Y 608.443,Z 130.189,A -85,B 0,C 180,E1 -519.018,E2 -519.018} C_VEL
LIN {X 0,Y 608.446,Z 130.198,A -85,B 0,C 180,E1 -521.828,E2 -521.828} C_VEL
LIN {X 0,Y 608.458,Z 130.187,A -85,B 0,C 180,E1 -524.594,E2 -524.594} C_VEL
LIN {X 0,Y 608.467,Z 130.191,A -85,B 0,C 180,E1 -527.323,E2 -527.323} C_VEL
LIN {X 0,Y 608.465,Z 130.189,A -85,B 0,C 180,E1 -530.023,E2 -530.023} C_VEL
LIN {X 0,Y 608.435,Z 130.191,A -85,B 0,C 180,E1 -532.7,E2 -532.7} C_VEL
LIN {X 0,Y 608.447,Z 130.189,A -85,B 0,C 180,E1 -534.698,E2 -534.698} C_VEL
LIN {X 0,Y 608.479,Z 130.194,A -85,B 0,C 180,E1 -537.352,E2 -537.352} C_VEL
LIN {X 0,Y 608.477,Z 130.185,A -85,B 0,C 180,E1 -540,E2 -540} C_VEL
LIN {X 0,Y 608.459,Z 130.189,A -85,B 0,C 180,E1 -542.648,E2 -542.648} C_VEL
LIN {X 0,Y 608.468,Z 130.192,A -85,B 0,C 180,E1 -545.302,E2 -545.302} C_VEL
LIN {X 0,Y 608.476,Z 130.185,A -85,B 0,C 180,E1 -547.967,E2 -547.967} C_VEL
LIN {X 0,Y 608.46,Z 130.189,A -85,B 0,C 180,E1 -549.446,E2 -549.446} C_VEL
LIN {X 0,Y 607.782,Z 130.274,A -85,B 0,C 180,E1 -549.999,E2 -549.999} C_VEL
LIN {X 0,Y 604.927,Z 130.637,A -85,B 0,C 180,E1 -550.896,E2 -550.896} C_VEL
LIN {X 0,Y 602.523,Z 130.931,A -85,B 0,C 180,E1 -551.617,E2 -551.617} C_VEL
LIN {X 0,Y 601.49,Z 131.056,A -85,B 0,C 180,E1 -552.174,E2 -552.174} C_VEL
LIN {X 0,Y 601.406,Z 131.068,A -85,B 0,C 180,E1 -552.362,E2 -552.362} C_VEL
LIN {X 0,Y 601.427,Z 131.071,A -85,B 0,C 180,E1 -554.897,E2 -554.897} C_VEL
LIN {X 0,Y 601.431,Z 131.068,A -85,B 0,C 180,E1 -556.986,E2 -556.986} C_VEL
LIN {X 0,Y 601.403,Z 131.066,A -85,B 0,C 180,E1 -559.81,E2 -559.81} C_VEL
LIN {X 0,Y 601.416,Z 131.074,A -85,B 0,C 180,E1 -562.606,E2 -562.606} C_VEL
LIN {X 0,Y 601.4,Z 131.07,A -85,B 0,C 180,E1 -564.879,E2 -564.879} C_VEL
LIN {X 0,Y 601.414,Z 131.064,A -85,B 0,C 180,E1 -567.362,E2 -567.362} C_VEL
LIN {X 0,Y 601.428,Z 131.07,A -85,B 0,C 180,E1 -570.164,E2 -570.164} C_VEL
LIN {X 0,Y 601.423,Z 131.066,A -85,B 0,C 180,E1 -572.716,E2 -572.716} C_VEL
LIN {X 0,Y 601.392,Z 131.067,A -85,B 0,C 180,E1 -575.112,E2 -575.112} C_VEL
LIN {X 0,Y 601.437,Z 131.063,A -85,B 0,C 180,E1 -577.419,E2 -577.419} C_VEL
LIN {X 0,Y 601.411,Z 131.075,A -85,B 0,C 180,E1 -579.995,E2 -579.995} C_VEL
LIN {X 0,Y 601.41,Z 131.066,A -85,B 0,C 180,E1 -582.671,E2 -582.671} C_VEL
LIN {X 0,Y 601.428,Z 131.067,A -85,B 0,C 180,E1 -585.482,E2 -585.482} C_VEL
LIN {X 0,Y 601.423,Z 131.065,A -85,B 0,C 180,E1 -588.407,E2 -588.407} C_VEL
LIN {X 0,Y 601.432,Z 131.07,A -85,B 0,C 180,E1 -591.529,E2 -591.529} C_VEL
LIN {X 0,Y 601.384,Z 131.07,A -85,B 0,C 180,E1 -594.245,E2 -594.245} C_VEL
LIN {X 0,Y 601.418,Z 131.064,A -85,B 0,C 180,E1 -596.686,E2 -596.686} C_VEL
LIN {X 0,Y 601.414,Z 131.068,A -85,B 0,C 180,E1 -599.058,E2 -599.058} C_VEL
LIN {X 0,Y 601.433,Z 131.072,A -85,B 0,C 180,E1 -601.373,E2 -601.373} C_VEL
LIN {X 0,Y 601.398,Z 131.072,A -85,B 0,C 180,E1 -603.636,E2 -603.636} C_VEL
LIN {X 0,Y 601.441,Z 131.063,A -85,B 0,C 180,E1 -605.859,E2 -605.859} C_VEL
LIN {X 0,Y 601.41,Z 131.069,A -85,B 0,C 180,E1 -608.761,E2 -608.761} C_VEL
LIN {X 0,Y 601.448,Z 131.166,A -85,B 0,C 180,E1 -610.348,E2 -610.348} C_VEL
LIN {X 0,Y 601.477,Z 146.22,A -85,B 0,C 180,E1 -612.84,E2 -612.84} C_VEL
LIN {X 0,Y 601.454,Z 162.207,A -85,B 0,C 180,E1 -615.45,E2 -615.45} C_VEL
LIN {X 0,Y 601.409,Z 171.067,A -85,B 0,C 180,E1 -616.882,E2 -616.882} C_VEL
LIN {X 0,Y 601.671,Z 177.127,A -85,B 0,C 180,E1 -616.963,E2 -616.963} C_VEL
LIN {X 0,Y 601.623,Z 277.824,A -85,B 0,C 180,E1 -618.183,E2 -618.183} C_VEL
LIN {X 0,Y 601.564,Z 290.374,A -85,B 0,C 180,E1 -618.459,E2 -618.459} C_VEL
LIN {X 0,Y 601.537,Z 303.567,A -85,B 0,C 180,E1 -618.895,E2 -618.895} C_VEL
LIN {X 0,Y 601.514,Z 314.75,A -85,B 0,C 180,E1 -619.396,E2 -619.396} C_VEL
LIN {X 0,Y 601.484,Z 326.523,A -85,B 0,C 180,E1 -620.076,E2 -620.076} C_VEL
LIN {X 0,Y 601.444,Z 337.033,A -85,B 0,C 180,E1 -620.839,E2 -620.839} C_VEL
LIN {X 0,Y 601.429,Z 345.64,A -85,B 0,C 180,E1 -621.601,E2 -621.601} C_VEL
LIN {X 0,Y 601.418,Z 353.568,A -85,B 0,C 180,E1 -622.446,E2 -622.446} C_VEL
LIN {X 0,Y 601.377,Z 360.89,A -85,B 0,C 180,E1 -623.393,E2 -623.393} C_VEL
LIN {X 0,Y 601.372,Z 366.612,A -85,B 0,C 180,E1 -624.299,E2 -624.299} C_VEL
LIN {X 0,Y 601.335,Z 371.753,A -85,B 0,C 180,E1 -625.307,E2 -625.307} C_VEL
LIN {X 0,Y 601.367,Z 375.743,A -85,B 0,C 180,E1 -626.315,E2 -626.315} C_VEL
LIN {X 0,Y 601.324,Z 378.693,A -85,B 0,C 180,E1 -627.32,E2 -627.32} C_VEL
LIN {X 0,Y 601.343,Z 380.127,A -85,B 0,C 180,E1 -627.991,E2 -627.991} C_VEL
LIN {X 0,Y 601.339,Z 381.753,A -85,B 0,C 180,E1 -629.33,E2 -629.33} C_VEL
LIN {X 0,Y 601.336,Z 381.996,A -85,B 0,C 180,E1 -630,E2 -630} C_VEL
LIN {X 0,Y 601.339,Z 381.815,A -85,B 0,C 180,E1 -630.67,E2 -630.67} C_VEL
LIN {X 0,Y 601.344,Z 380.276,A -85,B 0,C 180,E1 -632.009,E2 -632.009} C_VEL
LIN {X 0,Y 601.326,Z 378.916,A -85,B 0,C 180,E1 -632.68,E2 -632.68} C_VEL
LIN {X 0,Y 601.368,Z 376.04,A -85,B 0,C 180,E1 -633.685,E2 -633.685} C_VEL
LIN {X 0,Y 601.337,Z 372.141,A -85,B 0,C 180,E1 -634.693,E2 -634.693} C_VEL
LIN {X 0,Y 601.373,Z 367.11,A -85,B 0,C 180,E1 -635.701,E2 -635.701} C_VEL
LIN {X 0,Y 601.382,Z 360.792,A -85,B 0,C 180,E1 -636.711,E2 -636.711} C_VEL
LIN {X 0,Y 601.396,Z 352.875,A -85,B 0,C 180,E1 -637.723,E2 -637.723} C_VEL
LIN {X 0,Y 601.436,Z 343.03,A -85,B 0,C 180,E1 -638.738,E2 -638.738} C_VEL
LIN {X 0,Y 601.45,Z 332.71,A -85,B 0,C 180,E1 -639.585,E2 -639.585} C_VEL
LIN {X 0,Y 601.481,Z 321.089,A -85,B 0,C 180,E1 -640.349,E2 -640.349} C_VEL
LIN {X 0,Y 601.548,Z 309.895,A -85,B 0,C 180,E1 -640.928,E2 -640.928} C_VEL
LIN {X 0,Y 601.549,Z 297.315,A -85,B 0,C 180,E1 -641.421,E2 -641.421} C_VEL
LIN {X 0,Y 601.597,Z 284.54,A -85,B 0,C 180,E1 -641.775,E2 -641.775} C_VEL
LIN {X 0,Y 601.634,Z 272.256,A -85,B 0,C 180,E1 -641.988,E2 -641.988} C_VEL
LIN {X 0,Y 601.565,Z 172.107,A -85,B 0,C 180,E1 -643.19,E2 -643.19} C_VEL
LIN {X 0,Y 601.426,Z 171.026,A -85,B 0,C 180,E1 -643.214,E2 -643.214} C_VEL
LIN {X 0,Y 601.485,Z 154.232,A -85,B 0,C 180,E1 -645.937,E2 -645.937} C_VEL
LIN {X 0,Y 601.514,Z 136.549,A -85,B 0,C 180,E1 -648.845,E2 -648.845} C_VEL
LIN {X 0,Y 601.434,Z 131.065,A -85,B 0,C 180,E1 -649.764,E2 -649.764} C_VEL
LIN {X 0,Y 601.41,Z 131.073,A -85,B 0,C 180,E1 -652.683,E2 -652.683} C_VEL
LIN {X 0,Y 601.399,Z 131.076,A -85,B 0,C 180,E1 -654.879,E2 -654.879} C_VEL
LIN {X 0,Y 601.415,Z 131.066,A -85,B 0,C 180,E1 -657.362,E2 -657.362} C_VEL
LIN {X 0,Y 601.412,Z 131.065,A -85,B 0,C 180,E1 -659.393,E2 -659.393} C_VEL
LIN {X 0,Y 601.398,Z 131.067,A -85,B 0,C 180,E1 -661.727,E2 -661.727} C_VEL
LIN {X 0,Y 601.42,Z 131.068,A -85,B 0,C 180,E1 -664.119,E2 -664.119} C_VEL
LIN {X 0,Y 601.437,Z 131.062,A -85,B 0,C 180,E1 -667.382,E2 -667.382} C_VEL
LIN {X 0,Y 601.402,Z 131.071,A -85,B 0,C 180,E1 -669.996,E2 -669.996} C_VEL
LIN {X 0,Y 601.415,Z 131.068,A -85,B 0,C 180,E1 -672.67,E2 -672.67} C_VEL
LIN {X 0,Y 601.427,Z 131.064,A -85,B 0,C 180,E1 -675.482,E2 -675.482} C_VEL
LIN {X 0,Y 601.424,Z 131.068,A -85,B 0,C 180,E1 -678.407,E2 -678.407} C_VEL
LIN {X 0,Y 601.438,Z 131.062,A -85,B 0,C 180,E1 -680.875,E2 -680.875} C_VEL
LIN {X 0,Y 601.401,Z 131.069,A -85,B 0,C 180,E1 -683.417,E2 -683.417} C_VEL
LIN {X 0,Y 601.432,Z 131.069,A -85,B 0,C 180,E1 -686.064,E2 -686.064} C_VEL
LIN {X 0,Y 601.42,Z 131.064,A -85,B 0,C 180,E1 -688.545,E2 -688.545} C_VEL
LIN {X 0,Y 601.431,Z 131.067,A -85,B 0,C 180,E1 -691.373,E2 -691.373} C_VEL
LIN {X 0,Y 601.403,Z 131.076,A -85,B 0,C 180,E1 -693.636,E2 -693.636} C_VEL
LIN {X 0,Y 601.417,Z 131.064,A -85,B 0,C 180,E1 -696.589,E2 -696.589} C_VEL
LIN {X 0,Y 601.431,Z 131.072,A -85,B 0,C 180,E1 -699.478,E2 -699.478} C_VEL
LIN {X 0,Y 601.392,Z 131.067,A -85,B 0,C 180,E1 -702.311,E2 -702.311} C_VEL
LIN {X 0,Y 601.41,Z 131.065,A -85,B 0,C 180,E1 -704.409,E2 -704.409} C_VEL
LIN {X 0,Y 601.417,Z 131.074,A -85,B 0,C 180,E1 -707.172,E2 -707.172} C_VEL
LIN {X 0,Y 601.436,Z 131.062,A -85,B 0,C 180,E1 -709.905,E2 -709.905} C_VEL
LIN {X 0,Y 601.441,Z 131.065,A -85,B 0,C 180,E1 -712.615,E2 -712.615} C_VEL
LIN {X 0,Y 601.412,Z 131.069,A -85,B 0,C 180,E1 -715.308,E2 -715.308} C_VEL
LIN {X 0,Y 601.437,Z 131.062,A -85,B 0,C 180,E1 -717.991,E2 -717.991} C_VEL
LIN {X 0,Y 601.455,Z 131.068,A -85,B 0,C 180,E1 -720.669,E2 -720.669} C_VEL
LIN {X 0,Y 601.416,Z 131.066,A -85,B 0,C 180,E1 -723.35,E2 -723.35} C_VEL
LIN {X 0,Y 601.443,Z 131.063,A -85,B 0,C 180,E1 -726.037,E2 -726.037} C_VEL
LIN {X 0,Y 601.414,Z 131.072,A -85,B 0,C 180,E1 -728.738,E2 -728.738} C_VEL
LIN {X 0,Y 601.41,Z 131.065,A -85,B 0,C 180,E1 -731.459,E2 -731.459} C_VEL
LIN {X 0,Y 601.419,Z 131.071,A -85,B 0,C 180,E1 -734.205,E2 -734.205} C_VEL
LIN {X 0,Y 601.409,Z 131.066,A -85,B 0,C 180,E1 -736.987,E2 -736.987} C_VEL
LIN {X 0,Y 601.403,Z 131.07,A -85,B 0,C 180,E1 -739.81,E2 -739.81} C_VEL
LIN {X 0,Y 601.41,Z 131.067,A -85,B 0,C 180,E1 -742.683,E2 -742.683} C_VEL
LIN {X 0,Y 601.393,Z 131.067,A -85,B 0,C 180,E1 -744.879,E2 -744.879} C_VEL
LIN {X 0,Y 601.41,Z 131.067,A -85,B 0,C 180,E1 -747.362,E2 -747.362} C_VEL
LIN {X 0,Y 601.426,Z 131.069,A -85,B 0,C 180,E1 -750.164,E2 -750.164} C_VEL
LIN {X 0,Y 601.404,Z 131.066,A -85,B 0,C 180,E1 -752.713,E2 -752.713} C_VEL
LIN {X 0,Y 601.388,Z 131.069,A -85,B 0,C 180,E1 -755.111,E2 -755.111} C_VEL
LIN {X 0,Y 601.433,Z 131.068,A -85,B 0,C 180,E1 -757.419,E2 -757.419} C_VEL
LIN {X 0,Y 601.39,Z 131.071,A -85,B 0,C 180,E1 -759.997,E2 -759.997} C_VEL
LIN {X 0,Y 601.382,Z 131.069,A -85,B 0,C 180,E1 -762.673,E2 -762.673} C_VEL
LIN {X 0,Y 601.398,Z 131.076,A -85,B 0,C 180,E1 -765.48,E2 -765.48} C_VEL
LIN {X 0,Y 601.41,Z 131.065,A -85,B 0,C 180,E1 -768.409,E2 -768.409} C_VEL
LIN {X 0,Y 601.404,Z 131.07,A -85,B 0,C 180,E1 -770.873,E2 -770.873} C_VEL
LIN {X 0,Y 601.4,Z 131.072,A -85,B 0,C 180,E1 -773.417,E2 -773.417} C_VEL
LIN {X 0,Y 601.401,Z 131.066,A -85,B 0,C 180,E1 -776.069,E2 -776.069} C_VEL
LIN {X 0,Y 601.415,Z 131.067,A -85,B 0,C 180,E1 -778.547,E2 -778.547} C_VEL
LIN {X 0,Y 601.402,Z 131.07,A -85,B 0,C 180,E1 -781.372,E2 -781.372} C_VEL
LIN {X 0,Y 601.382,Z 131.069,A -85,B 0,C 180,E1 -783.635,E2 -783.635} C_VEL
LIN {X 0,Y 601.398,Z 131.067,A -85,B 0,C 180,E1 -785.857,E2 -785.857} C_VEL
LIN {X 0,Y 601.401,Z 131.152,A -85,B 0,C 180,E1 -787.779,E2 -787.779} C_VEL
LIN {X 0,Y 601.624,Z 137.919,A -85,B 0,C 180,E1 -788.769,E2 -788.769} C_VEL
LIN {X 0,Y 601.531,Z 156.136,A -85,B 0,C 180,E1 -791.377,E2 -791.377} C_VEL
LIN {X 0,Y 601.506,Z 175.172,A -85,B 0,C 180,E1 -794.063,E2 -794.063} C_VEL
LIN {X 0,Y 601.453,Z 195.149,A -85,B 0,C 180,E1 -796.829,E2 -796.829} C_VEL
LIN {X 0,Y 601.636,Z 255.964,A -85,B 0,C 180,E1 -797.562,E2 -797.562} C_VEL
LIN {X 0,Y 601.614,Z 302.951,A -85,B 0,C 180,E1 -798.14,E2 -798.14} C_VEL
LIN {X 0,Y 601.56,Z 316.22,A -85,B 0,C 180,E1 -798.438,E2 -798.438} C_VEL
LIN {X 0,Y 601.539,Z 327.945,A -85,B 0,C 180,E1 -798.827,E2 -798.827} C_VEL
LIN {X 0,Y 601.514,Z 338.926,A -85,B 0,C 180,E1 -799.311,E2 -799.311} C_VEL
LIN {X 0,Y 601.474,Z 349.582,A -85,B 0,C 180,E1 -799.906,E2 -799.906} C_VEL
LIN {X 0,Y 601.449,Z 360.477,A -85,B 0,C 180,E1 -800.669,E2 -800.669} C_VEL
LIN {X 0,Y 601.429,Z 371.113,A -85,B 0,C 180,E1 -801.601,E2 -801.601} C_VEL
LIN {X 0,Y 601.418,Z 378.961,A -85,B 0,C 180,E1 -802.446,E2 -802.446} C_VEL
LIN {X 0,Y 601.37,Z 386.225,A -85,B 0,C 180,E1 -803.398,E2 -803.398} C_VEL
LIN {X 0,Y 601.372,Z 391.866,A -85,B 0,C 180,E1 -804.299,E2 -804.299} C_VEL
LIN {X 0,Y 601.336,Z 396.95,A -85,B 0,C 180,E1 -805.307,E2 -805.307} C_VEL
LIN {X 0,Y 601.368,Z 400.896,A -85,B 0,C 180,E1 -806.315,E2 -806.315} C_VEL
LIN {X 0,Y 601.325,Z 403.809,A -85,B 0,C 180,E1 -807.32,E2 -807.32} C_VEL
LIN {X 0,Y 601.343,Z 405.202,A -85,B 0,C 180,E1 -807.991,E2 -807.991} C_VEL
LIN {X 0,Y 601.339,Z 406.784,A -85,B 0,C 180,E1 -809.33,E2 -809.33} C_VEL
LIN {X 0,Y 601.335,Z 407,A -85,B 0,C 180,E1 -810,E2 -810} C_VEL
LIN {X 0,Y 601.347,Z 406.184,A -85,B 0,C 180,E1 -811.339,E2 -811.339} C_VEL
LIN {X 0,Y 601.343,Z 405.202,A -85,B 0,C 180,E1 -812.009,E2 -812.009} C_VEL
LIN {X 0,Y 601.325,Z 403.809,A -85,B 0,C 180,E1 -812.68,E2 -812.68} C_VEL
LIN {X 0,Y 601.368,Z 400.896,A -85,B 0,C 180,E1 -813.685,E2 -813.685} C_VEL
LIN {X 0,Y 601.336,Z 396.95,A -85,B 0,C 180,E1 -814.693,E2 -814.693} C_VEL
LIN {X 0,Y 601.373,Z 390.877,A -85,B 0,C 180,E1 -815.869,E2 -815.869} C_VEL
LIN {X 0,Y 601.382,Z 384.236,A -85,B 0,C 180,E1 -816.88,E2 -816.88} C_VEL
LIN {X 0,Y 601.4,Z 375.99,A -85,B 0,C 180,E1 -817.892,E2 -817.892} C_VEL
LIN {X 0,Y 601.436,Z 367.537,A -85,B 0,C 180,E1 -818.738,E2 -818.738} C_VEL
LIN {X 0,Y 601.449,Z 357.093,A -85,B 0,C 180,E1 -819.585,E2 -819.585} C_VEL
LIN {X 0,Y 601.467,Z 346.758,A -85,B 0,C 180,E1 -820.264,E2 -820.264} C_VEL
LIN {X 0,Y 601.538,Z 334.597,A -85,B 0,C 180,E1 -820.896,E2 -820.896} C_VEL
LIN {X 0,Y 601.555,Z 322.218,A -85,B 0,C 180,E1 -821.379,E2 -821.379} C_VEL
LIN {X 0,Y 601.583,Z 309.438,A -85,B 0,C 180,E1 -821.733,E2 -821.733} C_VEL
LIN {X 0,Y 601.621,Z 297.085,A -85,B 0,C 180,E1 -821.946,E2 -821.946} C_VEL
LIN {X 0,Y 601.549,Z 196.037,A -85,B 0,C 180,E1 -823.158,E2 -823.158} C_VEL
LIN {X 0,Y 601.449,Z 194.884,A -85,B 0,C 180,E1 -823.193,E2 -823.193} C_VEL
LIN {X 0,Y 601.511,Z 173.93,A -85,B 0,C 180,E1 -826.111,E2 -826.111} C_VEL
LIN {X 0,Y 601.556,Z 154.486,A -85,B 0,C 180,E1 -828.857,E2 -828.857} C_VEL
LIN {X 0,Y 601.629,Z 134.193,A -85,B 0,C 180,E1 -831.771,E2 -831.771} C_VEL
LIN {X 0,Y 601.405,Z 131.069,A -85,B 0,C 180,E1 -832.265,E2 -832.265} C_VEL
LIN {X 0,Y 601.386,Z 131.074,A -85,B 0,C 180,E1 -834.879,E2 -834.879} C_VEL
LIN {X 0,Y 601.415,Z 131.07,A -85,B 0,C 180,E1 -837.362,E2 -837.362} C_VEL
LIN {X 0,Y 601.374,Z 131.069,A -85,B 0,C 180,E1 -840.167,E2 -840.167} C_VEL
LIN {X 0,Y 601.4,Z 131.073,A -85,B 0,C 180,E1 -842.712,E2 -842.712} C_VEL
LIN {X 0,Y 601.392,Z 131.073,A -85,B 0,C 180,E1 -845.111,E2 -845.111} C_VEL
LIN {X 0,Y 601.432,Z 131.064,A -85,B 0,C 180,E1 -847.419,E2 -847.419} C_VEL
LIN {X 0,Y 601.38,Z 131.069,A -85,B 0,C 180,E1 -849.997,E2 -849.997} C_VEL
LIN {X 0,Y 601.407,Z 131.076,A -85,B 0,C 180,E1 -852.671,E2 -852.671} C_VEL
LIN {X 0,Y 601.399,Z 131.066,A -85,B 0,C 180,E1 -855.479,E2 -855.479} C_VEL
LIN {X 0,Y 601.42,Z 131.073,A -85,B 0,C 180,E1 -858.407,E2 -858.407} C_VEL
LIN {X 0,Y 601.427,Z 131.066,A -85,B 0,C 180,E1 -860.875,E2 -860.875} C_VEL
LIN {X 0,Y 601.394,Z 131.067,A -85,B 0,C 180,E1 -863.416,E2 -863.416} C_VEL
LIN {X 0,Y 601.429,Z 131.07,A -85,B 0,C 180,E1 -866.065,E2 -866.065} C_VEL
LIN {X 0,Y 601.4,Z 131.066,A -85,B 0,C 180,E1 -869.057,E2 -869.057} C_VEL
LIN {X 0,Y 601.407,Z 131.066,A -85,B 0,C 180,E1 -871.372,E2 -871.372} C_VEL
LIN {X 0,Y 601.411,Z 131.073,A -85,B 0,C 180,E1 -874.133,E2 -874.133} C_VEL
LIN {X 0,Y 601.395,Z 131.068,A -85,B 0,C 180,E1 -876.589,E2 -876.589} C_VEL
LIN {X 0,Y 601.417,Z 131.068,A -85,B 0,C 180,E1 -879.478,E2 -879.478} C_VEL
LIN {X 0,Y 601.389,Z 131.07,A -85,B 0,C 180,E1 -882.311,E2 -882.311} C_VEL
LIN {X 0,Y 601.406,Z 131.066,A -85,B 0,C 180,E1 -884.408,E2 -884.408} C_VEL
LIN {X 0,Y 601.41,Z 131.068,A -85,B 0,C 180,E1 -887.172,E2 -887.172} C_VEL
LIN {X 0,Y 601.44,Z 131.065,A -85,B 0,C 180,E1 -889.905,E2 -889.905} C_VEL
LIN {X 0,Y 601.403,Z 131.066,A -85,B 0,C 180,E1 -892.614,E2 -892.614} C_VEL
LIN {X 0,Y 601.427,Z 131.072,A -85,B 0,C 180,E1 -895.308,E2 -895.308} C_VEL
LIN {X 0,Y 601.438,Z 131.062,A -85,B 0,C 180,E1 -897.991,E2 -897.991} C_VEL
LIN {X 0,Y 601.437,Z 131.064,A -85,B 0,C 180,E1 -900.67,E2 -900.67} C_VEL
LIN {X 0,Y 601.435,Z 131.068,A -85,B 0,C 180,E1 -903.35,E2 -903.35} C_VEL
LIN {X 0,Y 601.438,Z 131.061,A -85,B 0,C 180,E1 -906.037,E2 -906.037} C_VEL
LIN {X 0,Y 601.408,Z 131.072,A -85,B 0,C 180,E1 -908.738,E2 -908.738} C_VEL
LIN {X 0,Y 601.434,Z 131.064,A -85,B 0,C 180,E1 -911.458,E2 -911.458} C_VEL
LIN {X 0,Y 601.406,Z 131.068,A -85,B 0,C 180,E1 -912.362,E2 -912.362} C_VEL
LIN {X 0,Y 600.739,Z 131.158,A -85,B 0,C 180,E1 -912.922,E2 -912.922} C_VEL
LIN {X 0,Y 597.891,Z 131.514,A -85,B 0,C 180,E1 -913.83,E2 -913.83} C_VEL
LIN {X 0,Y 595.482,Z 131.812,A -85,B 0,C 180,E1 -914.56,E2 -914.56} C_VEL
LIN {X 0,Y 594.445,Z 131.938,A -85,B 0,C 180,E1 -915.124,E2 -915.124} C_VEL
LIN {X 0,Y 594.358,Z 131.946,A -85,B 0,C 180,E1 -915.314,E2 -915.314} C_VEL
LIN {X 0,Y 594.388,Z 131.943,A -85,B 0,C 180,E1 -917.194,E2 -917.194} C_VEL
LIN {X 0,Y 594.373,Z 131.943,A -85,B 0,C 180,E1 -920.054,E2 -920.054} C_VEL
LIN {X 0,Y 594.364,Z 131.946,A -85,B 0,C 180,E1 -922.967,E2 -922.967} C_VEL
LIN {X 0,Y 594.375,Z 131.942,A -85,B 0,C 180,E1 -925.193,E2 -925.193} C_VEL
LIN {X 0,Y 594.386,Z 131.94,A -85,B 0,C 180,E1 -927.527,E2 -927.527} C_VEL
LIN {X 0,Y 594.386,Z 131.951,A -85,B 0,C 180,E1 -930.328,E2 -930.328} C_VEL
LIN {X 0,Y 594.38,Z 131.942,A -85,B 0,C 180,E1 -932.95,E2 -932.95} C_VEL
LIN {X 0,Y 594.349,Z 131.945,A -85,B 0,C 180,E1 -935.409,E2 -935.409} C_VEL
LIN {X 0,Y 594.389,Z 131.947,A -85,B 0,C 180,E1 -937.941,E2 -937.941} C_VEL
LIN {X 0,Y 594.379,Z 131.941,A -85,B 0,C 180,E1 -940.822,E2 -940.822} C_VEL
LIN {X 0,Y 594.37,Z 131.951,A -85,B 0,C 180,E1 -943.84,E2 -943.84} C_VEL
LIN {X 0,Y 594.369,Z 131.942,A -85,B 0,C 180,E1 -946.701,E2 -946.701} C_VEL
LIN {X 0,Y 594.371,Z 131.947,A -85,B 0,C 180,E1 -949.433,E2 -949.433} C_VEL
LIN {X 0,Y 594.391,Z 131.94,A -85,B 0,C 180,E1 -952.392,E2 -952.392} C_VEL
LIN {X 0,Y 594.378,Z 131.949,A -85,B 0,C 180,E1 -955.42,E2 -955.42} C_VEL
LIN {X 0,Y 594.378,Z 131.941,A -85,B 0,C 180,E1 -958.358,E2 -958.358} C_VEL
LIN {X 0,Y 594.385,Z 131.944,A -85,B 0,C 180,E1 -961.042,E2 -961.042} C_VEL
LIN {X 0,Y 594.381,Z 131.942,A -85,B 0,C 180,E1 -963.979,E2 -963.979} C_VEL
LIN {X 0,Y 594.372,Z 131.942,A -85,B 0,C 180,E1 -966.295,E2 -966.295} C_VEL
LIN {X 0,Y 594.402,Z 131.948,A -85,B 0,C 180,E1 -969.224,E2 -969.224} C_VEL
LIN {X 0,Y 594.421,Z 132.102,A -85,B 0,C 180,E1 -970.263,E2 -970.263} C_VEL
LIN {X 0,Y 594.502,Z 145.158,A -85,B 0,C 180,E1 -972.455,E2 -972.455} C_VEL
LIN {X 0,Y 594.433,Z 162.211,A -85,B 0,C 180,E1 -975.274,E2 -975.274} C_VEL
LIN {X 0,Y 594.392,Z 171.07,A -85,B 0,C 180,E1 -976.724,E2 -976.724} C_VEL
LIN {X 0,Y 594.756,Z 175.384,A -85,B 0,C 180,E1 -976.787,E2 -976.787} C_VEL
LIN {X 0,Y 594.691,Z 277.853,A -85,B 0,C 180,E1 -978.043,E2 -978.043} C_VEL
LIN {X 0,Y 594.621,Z 291.152,A -85,B 0,C 180,E1 -978.344,E2 -978.344} C_VEL
LIN {X 0,Y 594.564,Z 303.049,A -85,B 0,C 180,E1 -978.743,E2 -978.743} C_VEL
LIN {X 0,Y 594.53,Z 314.764,A -85,B 0,C 180,E1 -979.27,E2 -979.27} C_VEL
LIN {X 0,Y 594.479,Z 326.53,A -85,B 0,C 180,E1 -979.958,E2 -979.958} C_VEL
LIN {X 0,Y 594.414,Z 337.042,A -85,B 0,C 180,E1 -980.73,E2 -980.73} C_VEL
LIN {X 0,Y 594.384,Z 345.646,A -85,B 0,C 180,E1 -981.501,E2 -981.501} C_VEL
LIN {X 0,Y 594.347,Z 353.573,A -85,B 0,C 180,E1 -982.355,E2 -982.355} C_VEL
LIN {X 0,Y 594.305,Z 361.395,A -85,B 0,C 180,E1 -983.39,E2 -983.39} C_VEL
LIN {X 0,Y 594.289,Z 368.441,A -85,B 0,C 180,E1 -984.571,E2 -984.571} C_VEL
LIN {X 0,Y 594.27,Z 373.183,A -85,B 0,C 180,E1 -985.591,E2 -985.591} C_VEL
LIN {X 0,Y 594.267,Z 376.817,A -85,B 0,C 180,E1 -986.61,E2 -986.61} C_VEL
LIN {X 0,Y 594.225,Z 378.695,A -85,B 0,C 180,E1 -987.288,E2 -987.288} C_VEL
LIN {X 0,Y 594.242,Z 380.127,A -85,B 0,C 180,E1 -987.967,E2 -987.967} C_VEL
LIN {X 0,Y 594.24,Z 381.753,A -85,B 0,C 180,E1 -989.322,E2 -989.322} C_VEL
LIN {X 0,Y 594.236,Z 381.996,A -85,B 0,C 180,E1 -990,E2 -990} C_VEL
LIN {X 0,Y 594.239,Z 381.815,A -85,B 0,C 180,E1 -990.678,E2 -990.678} C_VEL
LIN {X 0,Y 594.242,Z 380.275,A -85,B 0,C 180,E1 -992.033,E2 -992.033} C_VEL
LIN {X 0,Y 594.226,Z 378.914,A -85,B 0,C 180,E1 -992.712,E2 -992.712} C_VEL
LIN {X 0,Y 594.289,Z 376.038,A -85,B 0,C 180,E1 -993.729,E2 -993.729} C_VEL
LIN {X 0,Y 594.241,Z 372.138,A -85,B 0,C 180,E1 -994.749,E2 -994.749} C_VEL
LIN {X 0,Y 594.3,Z 367.107,A -85,B 0,C 180,E1 -995.769,E2 -995.769} C_VEL
LIN {X 0,Y 594.316,Z 360.788,A -85,B 0,C 180,E1 -996.791,E2 -996.791} C_VEL
LIN {X 0,Y 594.346,Z 352.87,A -85,B 0,C 180,E1 -997.815,E2 -997.815} C_VEL
LIN {X 0,Y 594.381,Z 343.024,A -85,B 0,C 180,E1 -998.842,E2 -998.842} C_VEL
LIN {X 0,Y 594.432,Z 332.704,A -85,B 0,C 180,E1 -999.699,E2 -999.699} C_VEL
LIN {X 0,Y 594.491,Z 321.078,A -85,B 0,C 180,E1 -1000.472,E2 -1000.472} C_VEL
LIN {X 0,Y 594.579,Z 309.072,A -85,B 0,C 180,E1 -1001.093,E2 -1001.093} C_VEL
LIN {X 0,Y 594.579,Z 296.234,A -85,B 0,C 180,E1 -1001.592,E2 -1001.592} C_VEL
LIN {X 0,Y 594.667,Z 283.6,A -85,B 0,C 180,E1 -1001.936,E2 -1001.936} C_VEL
LIN {X 0,Y 594.691,Z 270.457,A -85,B 0,C 180,E1 -1002.152,E2 -1002.152} C_VEL
LIN {X 0,Y 594.679,Z 172.958,A -85,B 0,C 180,E1 -1003.335,E2 -1003.335} C_VEL
LIN {X 0,Y 594.391,Z 171.022,A -85,B 0,C 180,E1 -1003.374,E2 -1003.374} C_VEL
LIN {X 0,Y 594.471,Z 153.162,A -85,B 0,C 180,E1 -1006.307,E2 -1006.307} C_VEL
LIN {X 0,Y 594.543,Z 136.424,A -85,B 0,C 180,E1 -1009.095,E2 -1009.095} C_VEL
LIN {X 0,Y 594.363,Z 131.947,A -85,B 0,C 180,E1 -1009.874,E2 -1009.874} C_VEL
LIN {X 0,Y 594.361,Z 131.952,A -85,B 0,C 180,E1 -1012.734,E2 -1012.734} C_VEL
LIN {X 0,Y 594.373,Z 131.946,A -85,B 0,C 180,E1 -1015.193,E2 -1015.193} C_VEL
LIN {X 0,Y 594.37,Z 131.942,A -85,B 0,C 180,E1 -1017.523,E2 -1017.523} C_VEL
LIN {X 0,Y 594.372,Z 131.947,A -85,B 0,C 180,E1 -1020.325,E2 -1020.325} C_VEL
LIN {X 0,Y 594.378,Z 131.945,A -85,B 0,C 180,E1 -1022.95,E2 -1022.95} C_VEL
LIN {X 0,Y 594.35,Z 131.945,A -85,B 0,C 180,E1 -1025.409,E2 -1025.409} C_VEL
LIN {X 0,Y 594.383,Z 131.943,A -85,B 0,C 180,E1 -1027.941,E2 -1027.941} C_VEL
LIN {X 0,Y 594.377,Z 131.944,A -85,B 0,C 180,E1 -1030.822,E2 -1030.822} C_VEL
LIN {X 0,Y 594.368,Z 131.942,A -85,B 0,C 180,E1 -1033.299,E2 -1033.299} C_VEL
LIN {X 0,Y 594.37,Z 131.952,A -85,B 0,C 180,E1 -1036.16,E2 -1036.16} C_VEL
LIN {X 0,Y 594.378,Z 131.941,A -85,B 0,C 180,E1 -1039.178,E2 -1039.178} C_VEL
LIN {X 0,Y 594.386,Z 131.949,A -85,B 0,C 180,E1 -1042.059,E2 -1042.059} C_VEL
LIN {X 0,Y 594.35,Z 131.945,A -85,B 0,C 180,E1 -1044.676,E2 -1044.676} C_VEL
LIN {X 0,Y 594.379,Z 131.942,A -85,B 0,C 180,E1 -1047.088,E2 -1047.088} C_VEL
LIN {X 0,Y 594.386,Z 131.949,A -85,B 0,C 180,E1 -1049.672,E2 -1049.672} C_VEL
LIN {X 0,Y 594.374,Z 131.942,A -85,B 0,C 180,E1 -1052.539,E2 -1052.539} C_VEL
LIN {X 0,Y 594.374,Z 131.942,A -85,B 0,C 180,E1 -1054.807,E2 -1054.807} C_VEL
LIN {X 0,Y 594.364,Z 131.949,A -85,B 0,C 180,E1 -1057.265,E2 -1057.265} C_VEL
LIN {X 0,Y 594.373,Z 131.944,A -85,B 0,C 180,E1 -1059.946,E2 -1059.946} C_VEL
LIN {X 0,Y 594.388,Z 131.942,A -85,B 0,C 180,E1 -1062.806,E2 -1062.806} C_VEL
LIN {X 0,Y 594.388,Z 131.942,A -85,B 0,C 180,E1 -1065.826,E2 -1065.826} C_VEL
LIN {X 0,Y 594.392,Z 131.94,A -85,B 0,C 180,E1 -1068.404,E2 -1068.404} C_VEL
LIN {X 0,Y 594.377,Z 131.95,A -85,B 0,C 180,E1 -1071.158,E2 -1071.158} C_VEL
LIN {X 0,Y 594.387,Z 131.94,A -85,B 0,C 180,E1 -1073.891,E2 -1073.891} C_VEL
LIN {X 0,Y 594.384,Z 131.945,A -85,B 0,C 180,E1 -1076.611,E2 -1076.611} C_VEL
LIN {X 0,Y 594.411,Z 131.94,A -85,B 0,C 180,E1 -1079.323,E2 -1079.323} C_VEL
LIN {X 0,Y 594.407,Z 131.938,A -85,B 0,C 180,E1 -1082.033,E2 -1082.033} C_VEL
LIN {X 0,Y 594.394,Z 131.948,A -85,B 0,C 180,E1 -1084.748,E2 -1084.748} C_VEL
LIN {X 0,Y 594.369,Z 131.942,A -85,B 0,C 180,E1 -1087.473,E2 -1087.473} C_VEL
LIN {X 0,Y 594.397,Z 131.944,A -85,B 0,C 180,E1 -1090.216,E2 -1090.216} C_VEL
LIN {X 0,Y 594.359,Z 131.945,A -85,B 0,C 180,E1 -1092.983,E2 -1092.983} C_VEL
LIN {X 0,Y 594.367,Z 131.943,A -85,B 0,C 180,E1 -1095.078,E2 -1095.078} C_VEL
LIN {X 0,Y 594.375,Z 131.941,A -85,B 0,C 180,E1 -1097.194,E2 -1097.194} C_VEL
LIN {X 0,Y 594.37,Z 131.95,A -85,B 0,C 180,E1 -1100.054,E2 -1100.054} C_VEL
LIN {X 0,Y 594.355,Z 131.944,A -85,B 0,C 180,E1 -1102.968,E2 -1102.968} C_VEL
LIN {X 0,Y 594.372,Z 131.942,A -85,B 0,C 180,E1 -1105.193,E2 -1105.193} C_VEL
LIN {X 0,Y 594.367,Z 131.946,A -85,B 0,C 180,E1 -1107.523,E2 -1107.523} C_VEL
LIN {X 0,Y 594.382,Z 131.944,A -85,B 0,C 180,E1 -1110.328,E2 -1110.328} C_VEL
LIN {X 0,Y 594.374,Z 131.942,A -85,B 0,C 180,E1 -1112.951,E2 -1112.951} C_VEL
LIN {X 0,Y 594.347,Z 131.95,A -85,B 0,C 180,E1 -1115.409,E2 -1115.409} C_VEL
LIN {X 0,Y 594.374,Z 131.947,A -85,B 0,C 180,E1 -1117.942,E2 -1117.942} C_VEL
LIN {X 0,Y 594.373,Z 131.942,A -85,B 0,C 180,E1 -1120.822,E2 -1120.822} C_VEL
LIN {X 0,Y 594.359,Z 131.948,A -85,B 0,C 180,E1 -1123.839,E2 -1123.839} C_VEL
LIN {X 0,Y 594.35,Z 131.945,A -85,B 0,C 180,E1 -1126.699,E2 -1126.699} C_VEL
LIN {X 0,Y 594.358,Z 131.952,A -85,B 0,C 180,E1 -1129.432,E2 -1129.432} C_VEL
LIN {X 0,Y 594.383,Z 131.941,A -85,B 0,C 180,E1 -1132.393,E2 -1132.393} C_VEL
LIN {X 0,Y 594.373,Z 131.947,A -85,B 0,C 180,E1 -1135.42,E2 -1135.42} C_VEL
LIN {X 0,Y 594.368,Z 131.943,A -85,B 0,C 180,E1 -1138.359,E2 -1138.359} C_VEL
LIN {X 0,Y 594.373,Z 131.95,A -85,B 0,C 180,E1 -1141.044,E2 -1141.044} C_VEL
LIN {X 0,Y 594.376,Z 131.945,A -85,B 0,C 180,E1 -1143.3,E2 -1143.3} C_VEL
LIN {X 0,Y 594.345,Z 131.949,A -85,B 0,C 180,E1 -1146.294,E2 -1146.294} C_VEL
LIN {X 0,Y 594.367,Z 131.988,A -85,B 0,C 180,E1 -1147.625,E2 -1147.625} C_VEL
LIN {X 0,Y 594.735,Z 136.677,A -85,B 0,C 180,E1 -1148.329,E2 -1148.329} C_VEL
LIN {X 0,Y 594.596,Z 155.956,A -85,B 0,C 180,E1 -1151.126,E2 -1151.126} C_VEL
LIN {X 0,Y 594.515,Z 175.172,A -85,B 0,C 180,E1 -1153.871,E2 -1153.871} C_VEL
LIN {X 0,Y 594.43,Z 195.149,A -85,B 0,C 180,E1 -1156.671,E2 -1156.671} C_VEL
LIN {X 0,Y 594.734,Z 202.303,A -85,B 0,C 180,E1 -1156.765,E2 -1156.765} C_VEL
LIN {X 0,Y 594.666,Z 302.95,A -85,B 0,C 180,E1 -1157.999,E2 -1157.999} C_VEL
LIN {X 0,Y 594.601,Z 316.221,A -85,B 0,C 180,E1 -1158.3,E2 -1158.3} C_VEL
LIN {X 0,Y 594.584,Z 329.365,A -85,B 0,C 180,E1 -1158.749,E2 -1158.749} C_VEL
LIN {X 0,Y 594.536,Z 340.633,A -85,B 0,C 180,E1 -1159.27,E2 -1159.27} C_VEL
LIN {X 0,Y 594.477,Z 352.202,A -85,B 0,C 180,E1 -1159.958,E2 -1159.958} C_VEL
LIN {X 0,Y 594.414,Z 362.598,A -85,B 0,C 180,E1 -1160.73,E2 -1160.73} C_VEL
LIN {X 0,Y 594.383,Z 371.113,A -85,B 0,C 180,E1 -1161.501,E2 -1161.501} C_VEL
LIN {X 0,Y 594.347,Z 378.961,A -85,B 0,C 180,E1 -1162.355,E2 -1162.355} C_VEL
LIN {X 0,Y 594.282,Z 386.813,A -85,B 0,C 180,E1 -1163.408,E2 -1163.408} C_VEL
LIN {X 0,Y 594.289,Z 393.681,A -85,B 0,C 180,E1 -1164.571,E2 -1164.571} C_VEL
LIN {X 0,Y 594.27,Z 398.372,A -85,B 0,C 180,E1 -1165.591,E2 -1165.591} C_VEL
LIN {X 0,Y 594.267,Z 401.957,A -85,B 0,C 180,E1 -1166.61,E2 -1166.61} C_VEL
LIN {X 0,Y 594.226,Z 403.809,A -85,B 0,C 180,E1 -1167.288,E2 -1167.288} C_VEL
LIN {X 0,Y 594.242,Z 405.201,A -85,B 0,C 180,E1 -1167.967,E2 -1167.967} C_VEL
LIN {X 0,Y 594.239,Z 406.784,A -85,B 0,C 180,E1 -1169.322,E2 -1169.322} C_VEL
LIN {X 0,Y 594.236,Z 407,A -85,B 0,C 180,E1 -1170,E2 -1170} C_VEL
LIN {X 0,Y 594.247,Z 406.185,A -85,B 0,C 180,E1 -1171.355,E2 -1171.355} C_VEL
LIN {X 0,Y 594.242,Z 405.201,A -85,B 0,C 180,E1 -1172.033,E2 -1172.033} C_VEL
LIN {X 0,Y 594.226,Z 403.81,A -85,B 0,C 180,E1 -1172.712,E2 -1172.712} C_VEL
LIN {X 0,Y 594.289,Z 400.896,A -85,B 0,C 180,E1 -1173.729,E2 -1173.729} C_VEL
LIN {X 0,Y 594.241,Z 396.949,A -85,B 0,C 180,E1 -1174.749,E2 -1174.749} C_VEL
LIN {X 0,Y 594.305,Z 390.877,A -85,B 0,C 180,E1 -1175.939,E2 -1175.939} C_VEL
LIN {X 0,Y 594.308,Z 384.236,A -85,B 0,C 180,E1 -1176.962,E2 -1176.962} C_VEL
LIN {X 0,Y 594.359,Z 375.99,A -85,B 0,C 180,E1 -1177.986,E2 -1177.986} C_VEL
LIN {X 0,Y 594.382,Z 367.538,A -85,B 0,C 180,E1 -1178.842,E2 -1178.842} C_VEL
LIN {X 0,Y 594.432,Z 357.095,A -85,B 0,C 180,E1 -1179.699,E2 -1179.699} C_VEL
LIN {X 0,Y 594.481,Z 346.758,A -85,B 0,C 180,E1 -1180.386,E2 -1180.386} C_VEL
LIN {X 0,Y 594.558,Z 335.724,A -85,B 0,C 180,E1 -1180.973,E2 -1180.973} C_VEL
LIN {X 0,Y 594.579,Z 323.712,A -85,B 0,C 180,E1 -1181.464,E2 -1181.464} C_VEL
LIN {X 0,Y 594.625,Z 310.351,A -85,B 0,C 180,E1 -1181.85,E2 -1181.85} C_VEL
LIN {X 0,Y 594.699,Z 297.085,A -85,B 0,C 180,E1 -1182.087,E2 -1182.087} C_VEL
LIN {X 0,Y 594.693,Z 197.057,A -85,B 0,C 180,E1 -1183.3,E2 -1183.3} C_VEL
LIN {X 0,Y 594.424,Z 194.884,A -85,B 0,C 180,E1 -1183.351,E2 -1183.351} C_VEL
LIN {X 0,Y 594.5,Z 173.93,A -85,B 0,C 180,E1 -1186.306,E2 -1186.306} C_VEL
LIN {X 0,Y 594.587,Z 155.185,A -85,B 0,C 180,E1 -1188.985,E2 -1188.985} C_VEL
LIN {X 0,Y 594.736,Z 136.677,A -85,B 0,C 180,E1 -1191.671,E2 -1191.671} C_VEL
LIN {X 0,Y 594.377,Z 131.946,A -85,B 0,C 180,E1 -1192.393,E2 -1192.393} C_VEL
LIN {X 0,Y 594.364,Z 131.953,A -85,B 0,C 180,E1 -1195.194,E2 -1195.194} C_VEL
LIN {X 0,Y 594.349,Z 131.948,A -85,B 0,C 180,E1 -1197.519,E2 -1197.519} C_VEL
LIN {X 0,Y 594.338,Z 131.946,A -85,B 0,C 180,E1 -1199.778,E2 -1199.778} C_VEL
LIN {X 0,Y 594.345,Z 131.945,A -85,B 0,C 180,E1 -1202.148,E2 -1202.148} C_VEL
LIN {X 0,Y 594.373,Z 131.947,A -85,B 0,C 180,E1 -1204.58,E2 -1204.58} C_VEL
LIN {X 0,Y 594.383,Z 131.941,A -85,B 0,C 180,E1 -1207.607,E2 -1207.607} C_VEL
LIN {X 0,Y 594.359,Z 131.951,A -85,B 0,C 180,E1 -1210.568,E2 -1210.568} C_VEL
LIN {X 0,Y 594.35,Z 131.945,A -85,B 0,C 180,E1 -1213.301,E2 -1213.301} C_VEL
LIN {X 0,Y 594.359,Z 131.947,A -85,B 0,C 180,E1 -1216.161,E2 -1216.161} C_VEL
LIN {X 0,Y 594.374,Z 131.942,A -85,B 0,C 180,E1 -1219.178,E2 -1219.178} C_VEL
LIN {X 0,Y 594.374,Z 131.947,A -85,B 0,C 180,E1 -1222.058,E2 -1222.058} C_VEL
LIN {X 0,Y 594.349,Z 131.949,A -85,B 0,C 180,E1 -1224.677,E2 -1224.677} C_VEL
LIN {X 0,Y 594.373,Z 131.942,A -85,B 0,C 180,E1 -1227.089,E2 -1227.089} C_VEL
LIN {X 0,Y 594.367,Z 131.945,A -85,B 0,C 180,E1 -1229.675,E2 -1229.675} C_VEL
LIN {X 0,Y 594.375,Z 131.944,A -85,B 0,C 180,E1 -1232.539,E2 -1232.539} C_VEL
LIN {X 0,Y 594.398,Z 131.942,A -85,B 0,C 180,E1 -1235.564,E2 -1235.564} C_VEL
LIN {X 0,Y 594.361,Z 131.945,A -85,B 0,C 180,E1 -1238.496,E2 -1238.496} C_VEL
LIN {X 0,Y 594.377,Z 131.945,A -85,B 0,C 180,E1 -1241.382,E2 -1241.382} C_VEL
LIN {X 0,Y 594.361,Z 131.945,A -85,B 0,C 180,E1 -1244.219,E2 -1244.219} C_VEL
LIN {X 0,Y 594.376,Z 131.942,A -85,B 0,C 180,E1 -1246.321,E2 -1246.321} C_VEL
LIN {X 0,Y 594.372,Z 131.945,A -85,B 0,C 180,E1 -1249.095,E2 -1249.095} C_VEL
LIN {X 0,Y 594.414,Z 131.941,A -85,B 0,C 180,E1 -1251.843,E2 -1251.843} C_VEL
LIN {X 0,Y 594.385,Z 131.94,A -85,B 0,C 180,E1 -1254.572,E2 -1254.572} C_VEL
LIN {X 0,Y 594.409,Z 131.947,A -85,B 0,C 180,E1 -1257.289,E2 -1257.289} C_VEL
LIN {X 0,Y 594.414,Z 131.937,A -85,B 0,C 180,E1 -1260,E2 -1260} C_VEL
LIN {X 0,Y 594.395,Z 131.942,A -85,B 0,C 180,E1 -1262.711,E2 -1262.711} C_VEL
LIN {X 0,Y 594.4,Z 131.943,A -85,B 0,C 180,E1 -1265.428,E2 -1265.428} C_VEL
LIN {X 0,Y 594.411,Z 131.937,A -85,B 0,C 180,E1 -1268.157,E2 -1268.157} C_VEL
LIN {X 0,Y 594.388,Z 131.947,A -85,B 0,C 180,E1 -1271.074,E2 -1271.074} C_VEL
LIN {X 0,Y 594.382,Z 131.941,A -85,B 0,C 180,E1 -1273.679,E2 -1273.679} C_VEL
LIN {X 0,Y 594.358,Z 131.946,A -85,B 0,C 180,E1 -1275.314,E2 -1275.314} C_VEL
LIN {X 0,Y 593.683,Z 132.029,A -85,B 0,C 180,E1 -1275.88,E2 -1275.88} C_VEL
LIN {X 0,Y 590.817,Z 132.394,A -85,B 0,C 180,E1 -1276.798,E2 -1276.798} C_VEL
LIN {X 0,Y 588.407,Z 132.69,A -85,B 0,C 180,E1 -1277.537,E2 -1277.537} C_VEL
LIN {X 0,Y 587.386,Z 132.814,A -85,B 0,C 180,E1 -1278.107,E2 -1278.107} C_VEL
LIN {X 0,Y 587.309,Z 132.824,A -85,B 0,C 180,E1 -1278.3,E2 -1278.3} C_VEL
LIN {X 0,Y 587.331,Z 132.822,A -85,B 0,C 180,E1 -1281.038,E2 -1281.038} C_VEL
LIN {X 0,Y 587.321,Z 132.821,A -85,B 0,C 180,E1 -1283.259,E2 -1283.259} C_VEL
LIN {X 0,Y 587.334,Z 132.818,A -85,B 0,C 180,E1 -1285.517,E2 -1285.517} C_VEL
LIN {X 0,Y 587.348,Z 132.819,A -85,B 0,C 180,E1 -1287.818,E2 -1287.818} C_VEL
LIN {X 0,Y 587.336,Z 132.825,A -85,B 0,C 180,E1 -1290.51,E2 -1290.51} C_VEL
LIN {X 0,Y 587.335,Z 132.819,A -85,B 0,C 180,E1 -1293.397,E2 -1293.397} C_VEL
LIN {X 0,Y 587.291,Z 132.83,A -85,B 0,C 180,E1 -1295.9,E2 -1295.9} C_VEL
LIN {X 0,Y 587.334,Z 132.822,A -85,B 0,C 180,E1 -1298.479,E2 -1298.479} C_VEL
LIN {X 0,Y 587.338,Z 132.818,A -85,B 0,C 180,E1 -1301.157,E2 -1301.157} C_VEL
LIN {X 0,Y 587.328,Z 132.826,A -85,B 0,C 180,E1 -1304.114,E2 -1304.114} C_VEL
LIN {X 0,Y 587.317,Z 132.821,A -85,B 0,C 180,E1 -1306.994,E2 -1306.994} C_VEL
LIN {X 0,Y 587.314,Z 132.831,A -85,B 0,C 180,E1 -1309.746,E2 -1309.746} C_VEL
LIN {X 0,Y 587.346,Z 132.818,A -85,B 0,C 180,E1 -1312.393,E2 -1312.393} C_VEL
LIN {X 0,Y 587.343,Z 132.826,A -85,B 0,C 180,E1 -1315.654,E2 -1315.654} C_VEL
LIN {X 0,Y 587.342,Z 132.818,A -85,B 0,C 180,E1 -1318.231,E2 -1318.231} C_VEL
LIN {X 0,Y 587.351,Z 132.819,A -85,B 0,C 180,E1 -1320.867,E2 -1320.867} C_VEL
LIN {X 0,Y 587.341,Z 132.821,A -85,B 0,C 180,E1 -1323.823,E2 -1323.823} C_VEL
LIN {X 0,Y 587.318,Z 132.822,A -85,B 0,C 180,E1 -1325.993,E2 -1325.993} C_VEL
LIN {X 0,Y 587.319,Z 132.821,A -85,B 0,C 180,E1 -1328.226,E2 -1328.226} C_VEL
LIN {X 0,Y 587.393,Z 132.905,A -85,B 0,C 180,E1 -1330.154,E2 -1330.154} C_VEL
LIN {X 0,Y 587.503,Z 143.029,A -85,B 0,C 180,E1 -1331.879,E2 -1331.879} C_VEL
LIN {X 0,Y 587.407,Z 160.082,A -85,B 0,C 180,E1 -1334.739,E2 -1334.739} C_VEL
LIN {X 0,Y 587.369,Z 171.184,A -85,B 0,C 180,E1 -1336.565,E2 -1336.565} C_VEL
LIN {X 0,Y 587.854,Z 175.429,A -85,B 0,C 180,E1 -1336.629,E2 -1336.629} C_VEL
LIN {X 0,Y 587.743,Z 277.883,A -85,B 0,C 180,E1 -1337.899,E2 -1337.899} C_VEL
LIN {X 0,Y 587.669,Z 291.171,A -85,B 0,C 180,E1 -1338.204,E2 -1338.204} C_VEL
LIN {X 0,Y 587.612,Z 303.733,A -85,B 0,C 180,E1 -1338.634,E2 -1338.634} C_VEL
LIN {X 0,Y 587.548,Z 314.777,A -85,B 0,C 180,E1 -1339.141,E2 -1339.141} C_VEL
LIN {X 0,Y 587.468,Z 326.536,A -85,B 0,C 180,E1 -1339.837,E2 -1339.837} C_VEL
LIN {X 0,Y 587.394,Z 337.05,A -85,B 0,C 180,E1 -1340.618,E2 -1340.618} C_VEL
LIN {X 0,Y 587.323,Z 345.652,A -85,B 0,C 180,E1 -1341.398,E2 -1341.398} C_VEL
LIN {X 0,Y 587.274,Z 353.577,A -85,B 0,C 180,E1 -1342.263,E2 -1342.263} C_VEL
LIN {X 0,Y 587.236,Z 360.148,A -85,B 0,C 180,E1 -1343.126,E2 -1343.126} C_VEL
LIN {X 0,Y 587.237,Z 366.618,A -85,B 0,C 180,E1 -1344.161,E2 -1344.161} C_VEL
LIN {X 0,Y 587.146,Z 371.758,A -85,B 0,C 180,E1 -1345.194,E2 -1345.194} C_VEL
LIN {X 0,Y 587.213,Z 375.748,A -85,B 0,C 180,E1 -1346.226,E2 -1346.226} C_VEL
LIN {X 0,Y 587.131,Z 378.697,A -85,B 0,C 180,E1 -1347.256,E2 -1347.256} C_VEL
LIN {X 0,Y 587.141,Z 380.127,A -85,B 0,C 180,E1 -1347.942,E2 -1347.942} C_VEL
LIN {X 0,Y 587.14,Z 381.754,A -85,B 0,C 180,E1 -1349.314,E2 -1349.314} C_VEL
LIN {X 0,Y 587.137,Z 381.996,A -85,B 0,C 180,E1 -1350,E2 -1350} C_VEL
LIN {X 0,Y 587.14,Z 381.815,A -85,B 0,C 180,E1 -1350.686,E2 -1350.686} C_VEL
LIN {X 0,Y 587.141,Z 380.273,A -85,B 0,C 180,E1 -1352.058,E2 -1352.058} C_VEL
LIN {X 0,Y 587.133,Z 378.912,A -85,B 0,C 180,E1 -1352.744,E2 -1352.744} C_VEL
LIN {X 0,Y 587.213,Z 376.036,A -85,B 0,C 180,E1 -1353.774,E2 -1353.774} C_VEL
LIN {X 0,Y 587.147,Z 372.136,A -85,B 0,C 180,E1 -1354.806,E2 -1354.806} C_VEL
LIN {X 0,Y 587.23,Z 367.105,A -85,B 0,C 180,E1 -1355.839,E2 -1355.839} C_VEL
LIN {X 0,Y 587.23,Z 360.784,A -85,B 0,C 180,E1 -1356.874,E2 -1356.874} C_VEL
LIN {X 0,Y 587.288,Z 352.865,A -85,B 0,C 180,E1 -1357.91,E2 -1357.91} C_VEL
LIN {X 0,Y 587.343,Z 343.017,A -85,B 0,C 180,E1 -1358.949,E2 -1358.949} C_VEL
LIN {X 0,Y 587.419,Z 332.699,A -85,B 0,C 180,E1 -1359.816,E2 -1359.816} C_VEL
LIN {X 0,Y 587.497,Z 321.066,A -85,B 0,C 180,E1 -1360.598,E2 -1360.598} C_VEL
LIN {X 0,Y 587.607,Z 309.934,A -85,B 0,C 180,E1 -1361.188,E2 -1361.188} C_VEL
LIN {X 0,Y 587.625,Z 297.436,A -85,B 0,C 180,E1 -1361.69,E2 -1361.69} C_VEL
LIN {X 0,Y 587.709,Z 284.492,A -85,B 0,C 180,E1 -1362.058,E2 -1362.058} C_VEL
LIN {X 0,Y 587.773,Z 272.177,A -85,B 0,C 180,E1 -1362.275,E2 -1362.275} C_VEL
LIN {X 0,Y 587.774,Z 173.805,A -85,B 0,C 180,E1 -1363.483,E2 -1363.483} C_VEL
LIN {X 0,Y 587.372,Z 171.019,A -85,B 0,C 180,E1 -1363.537,E2 -1363.537} C_VEL
LIN {X 0,Y 587.462,Z 153.159,A -85,B 0,C 180,E1 -1366.507,E2 -1366.507} C_VEL
LIN {X 0,Y 587.552,Z 136.739,A -85,B 0,C 180,E1 -1369.277,E2 -1369.277} C_VEL
LIN {X 0,Y 587.324,Z 132.825,A -85,B 0,C 180,E1 -1369.985,E2 -1369.985} C_VEL
LIN {X 0,Y 587.313,Z 132.831,A -85,B 0,C 180,E1 -1372.866,E2 -1372.866} C_VEL
LIN {X 0,Y 587.33,Z 132.82,A -85,B 0,C 180,E1 -1375.517,E2 -1375.517} C_VEL
LIN {X 0,Y 587.341,Z 132.818,A -85,B 0,C 180,E1 -1377.818,E2 -1377.818} C_VEL
LIN {X 0,Y 587.327,Z 132.827,A -85,B 0,C 180,E1 -1380.508,E2 -1380.508} C_VEL
LIN {X 0,Y 587.338,Z 132.82,A -85,B 0,C 180,E1 -1383.111,E2 -1383.111} C_VEL
LIN {X 0,Y 587.291,Z 132.826,A -85,B 0,C 180,E1 -1385.9,E2 -1385.9} C_VEL
LIN {X 0,Y 587.329,Z 132.828,A -85,B 0,C 180,E1 -1388.479,E2 -1388.479} C_VEL
LIN {X 0,Y 587.336,Z 132.818,A -85,B 0,C 180,E1 -1391.157,E2 -1391.157} C_VEL
LIN {X 0,Y 587.328,Z 132.828,A -85,B 0,C 180,E1 -1394.113,E2 -1394.113} C_VEL
LIN {X 0,Y 587.314,Z 132.821,A -85,B 0,C 180,E1 -1396.993,E2 -1396.993} C_VEL
LIN {X 0,Y 587.318,Z 132.826,A -85,B 0,C 180,E1 -1399.746,E2 -1399.746} C_VEL
LIN {X 0,Y 587.346,Z 132.82,A -85,B 0,C 180,E1 -1402.392,E2 -1402.392} C_VEL
LIN {X 0,Y 587.359,Z 132.824,A -85,B 0,C 180,E1 -1405.78,E2 -1405.78} C_VEL
LIN {X 0,Y 587.341,Z 132.821,A -85,B 0,C 180,E1 -1408.231,E2 -1408.231} C_VEL
LIN {X 0,Y 587.349,Z 132.817,A -85,B 0,C 180,E1 -1410.866,E2 -1410.866} C_VEL
LIN {X 0,Y 587.36,Z 132.822,A -85,B 0,C 180,E1 -1413.819,E2 -1413.819} C_VEL
LIN {X 0,Y 587.335,Z 132.822,A -85,B 0,C 180,E1 -1415.993,E2 -1415.993} C_VEL
LIN {X 0,Y 587.324,Z 132.82,A -85,B 0,C 180,E1 -1418.226,E2 -1418.226} C_VEL
LIN {X 0,Y 587.351,Z 132.822,A -85,B 0,C 180,E1 -1421.151,E2 -1421.151} C_VEL
LIN {X 0,Y 587.322,Z 132.821,A -85,B 0,C 180,E1 -1424.025,E2 -1424.025} C_VEL
LIN {X 0,Y 587.358,Z 132.815,A -85,B 0,C 180,E1 -1426.154,E2 -1426.154} C_VEL
LIN {X 0,Y 587.341,Z 132.825,A -85,B 0,C 180,E1 -1428.962,E2 -1428.962} C_VEL
LIN {X 0,Y 587.363,Z 132.816,A -85,B 0,C 180,E1 -1431.745,E2 -1431.745} C_VEL
LIN {X 0,Y 587.363,Z 132.818,A -85,B 0,C 180,E1 -1434.507,E2 -1434.507} C_VEL
LIN {X 0,Y 587.366,Z 132.819,A -85,B 0,C 180,E1 -1437.257,E2 -1437.257} C_VEL
LIN {X 0,Y 587.383,Z 132.813,A -85,B 0,C 180,E1 -1440,E2 -1440} C_VEL
LIN {X 0,Y 587.373,Z 132.824,A -85,B 0,C 180,E1 -1442.743,E2 -1442.743} C_VEL
LIN {X 0,Y 587.355,Z 132.816,A -85,B 0,C 180,E1 -1445.493,E2 -1445.493} C_VEL
LIN {X 0,Y 587.366,Z 132.82,A -85,B 0,C 180,E1 -1448.255,E2 -1448.255} C_VEL
LIN {X 0,Y 587.347,Z 132.818,A -85,B 0,C 180,E1 -1451.134,E2 -1451.134} C_VEL
LIN {X 0,Y 587.364,Z 132.823,A -85,B 0,C 180,E1 -1454.26,E2 -1454.26} C_VEL
LIN {X 0,Y 587.34,Z 132.818,A -85,B 0,C 180,E1 -1457.406,E2 -1457.406} C_VEL
LIN {X 0,Y 587.323,Z 132.828,A -85,B 0,C 180,E1 -1460.305,E2 -1460.305} C_VEL
LIN {X 0,Y 587.314,Z 132.821,A -85,B 0,C 180,E1 -1463.259,E2 -1463.259} C_VEL
LIN {X 0,Y 587.331,Z 132.821,A -85,B 0,C 180,E1 -1465.517,E2 -1465.517} C_VEL
LIN {X 0,Y 587.336,Z 132.826,A -85,B 0,C 180,E1 -1467.818,E2 -1467.818} C_VEL
LIN {X 0,Y 587.33,Z 132.82,A -85,B 0,C 180,E1 -1470.509,E2 -1470.509} C_VEL
LIN {X 0,Y 587.332,Z 132.822,A -85,B 0,C 180,E1 -1473.397,E2 -1473.397} C_VEL
LIN {X 0,Y 587.287,Z 132.831,A -85,B 0,C 180,E1 -1475.9,E2 -1475.9} C_VEL
LIN {X 0,Y 587.319,Z 132.821,A -85,B 0,C 180,E1 -1478.48,E2 -1478.48} C_VEL
LIN {X 0,Y 587.334,Z 132.822,A -85,B 0,C 180,E1 -1481.157,E2 -1481.157} C_VEL
LIN {X 0,Y 587.311,Z 132.823,A -85,B 0,C 180,E1 -1484.112,E2 -1484.112} C_VEL
LIN {X 0,Y 587.305,Z 132.826,A -85,B 0,C 180,E1 -1486.993,E2 -1486.993} C_VEL
LIN {X 0,Y 587.304,Z 132.825,A -85,B 0,C 180,E1 -1489.745,E2 -1489.745} C_VEL
LIN {X 0,Y 587.339,Z 132.818,A -85,B 0,C 180,E1 -1492.392,E2 -1492.392} C_VEL
LIN {X 0,Y 587.322,Z 132.827,A -85,B 0,C 180,E1 -1494.944,E2 -1494.944} C_VEL
LIN {X 0,Y 587.327,Z 132.824,A -85,B 0,C 180,E1 -1497.42,E2 -1497.42} C_VEL
LIN {X 0,Y 587.296,Z 132.824,A -85,B 0,C 180,E1 -1499.828,E2 -1499.828} C_VEL
LIN {X 0,Y 587.301,Z 132.825,A -85,B 0,C 180,E1 -1502.317,E2 -1502.317} C_VEL
LIN {X 0,Y 587.299,Z 132.828,A -85,B 0,C 180,E1 -1505.239,E2 -1505.239} C_VEL
LIN {X 0,Y 587.344,Z 132.877,A -85,B 0,C 180,E1 -1507.487,E2 -1507.487} C_VEL
LIN {X 0,Y 587.804,Z 137.915,A -85,B 0,C 180,E1 -1508.245,E2 -1508.245} C_VEL
LIN {X 0,Y 587.639,Z 155.846,A -85,B 0,C 180,E1 -1510.878,E2 -1510.878} C_VEL
LIN {X 0,Y 587.518,Z 173.93,A -85,B 0,C 180,E1 -1513.495,E2 -1513.495} C_VEL
LIN {X 0,Y 587.405,Z 194.419,A -85,B 0,C 180,E1 -1516.42,E2 -1516.42} C_VEL
LIN {X 0,Y 587.387,Z 195.149,A -85,B 0,C 180,E1 -1516.508,E2 -1516.508} C_VEL
LIN {X 0,Y 587.852,Z 200.515,A -85,B 0,C 180,E1 -1516.585,E2 -1516.585} C_VEL
LIN {X 0,Y 587.727,Z 302.95,A -85,B 0,C 180,E1 -1517.855,E2 -1517.855} C_VEL
LIN {X 0,Y 587.668,Z 316.222,A -85,B 0,C 180,E1 -1518.16,E2 -1518.16} C_VEL
LIN {X 0,Y 587.602,Z 328.689,A -85,B 0,C 180,E1 -1518.587,E2 -1518.587} C_VEL
LIN {X 0,Y 587.536,Z 340.631,A -85,B 0,C 180,E1 -1519.141,E2 -1519.141} C_VEL
LIN {X 0,Y 587.464,Z 352.204,A -85,B 0,C 180,E1 -1519.837,E2 -1519.837} C_VEL
LIN {X 0,Y 587.394,Z 362.6,A -85,B 0,C 180,E1 -1520.618,E2 -1520.618} C_VEL
LIN {X 0,Y 587.321,Z 371.113,A -85,B 0,C 180,E1 -1521.398,E2 -1521.398} C_VEL
LIN {X 0,Y 587.274,Z 378.961,A -85,B 0,C 180,E1 -1522.263,E2 -1522.263} C_VEL
LIN {X 0,Y 587.23,Z 385.469,A -85,B 0,C 180,E1 -1523.126,E2 -1523.126} C_VEL
LIN {X 0,Y 587.237,Z 391.867,A -85,B 0,C 180,E1 -1524.161,E2 -1524.161} C_VEL
LIN {X 0,Y 587.147,Z 396.95,A -85,B 0,C 180,E1 -1525.194,E2 -1525.194} C_VEL
LIN {X 0,Y 587.213,Z 400.896,A -85,B 0,C 180,E1 -1526.226,E2 -1526.226} C_VEL
LIN {X 0,Y 587.132,Z 403.809,A -85,B 0,C 180,E1 -1527.256,E2 -1527.256} C_VEL
LIN {X 0,Y 587.141,Z 405.199,A -85,B 0,C 180,E1 -1527.942,E2 -1527.942} C_VEL
LIN {X 0,Y 587.14,Z 406.785,A -85,B 0,C 180,E1 -1529.314,E2 -1529.314} C_VEL
LIN {X 0,Y 587.137,Z 407,A -85,B 0,C 180,E1 -1530,E2 -1530} C_VEL
LIN {X 0,Y 587.147,Z 406.186,A -85,B 0,C 180,E1 -1531.372,E2 -1531.372} C_VEL
LIN {X 0,Y 587.141,Z 405.2,A -85,B 0,C 180,E1 -1532.058,E2 -1532.058} C_VEL
LIN {X 0,Y 587.132,Z 403.81,A -85,B 0,C 180,E1 -1532.744,E2 -1532.744} C_VEL
LIN {X 0,Y 587.213,Z 400.896,A -85,B 0,C 180,E1 -1533.774,E2 -1533.774} C_VEL
LIN {X 0,Y 587.147,Z 396.949,A -85,B 0,C 180,E1 -1534.806,E2 -1534.806} C_VEL
LIN {X 0,Y 587.218,Z 390.877,A -85,B 0,C 180,E1 -1536.011,E2 -1536.011} C_VEL
LIN {X 0,Y 587.245,Z 384.237,A -85,B 0,C 180,E1 -1537.046,E2 -1537.046} C_VEL
LIN {X 0,Y 587.299,Z 375.99,A -85,B 0,C 180,E1 -1538.083,E2 -1538.083} C_VEL
LIN {X 0,Y 587.343,Z 367.538,A -85,B 0,C 180,E1 -1538.949,E2 -1538.949} C_VEL
LIN {X 0,Y 587.419,Z 357.097,A -85,B 0,C 180,E1 -1539.816,E2 -1539.816} C_VEL
LIN {X 0,Y 587.497,Z 346.756,A -85,B 0,C 180,E1 -1540.511,E2 -1540.511} C_VEL
LIN {X 0,Y 587.561,Z 334.817,A -85,B 0,C 180,E1 -1541.149,E2 -1541.149} C_VEL
LIN {X 0,Y 587.629,Z 322.599,A -85,B 0,C 180,E1 -1541.639,E2 -1541.639} C_VEL
LIN {X 0,Y 587.705,Z 309.435,A -85,B 0,C 180,E1 -1542.014,E2 -1542.014} C_VEL
LIN {X 0,Y 587.769,Z 297.085,A -85,B 0,C 180,E1 -1542.232,E2 -1542.232} C_VEL
LIN {X 0,Y 587.703,Z 196.934,A -85,B 0,C 180,E1 -1543.463,E2 -1543.463} C_VEL
LIN {X 0,Y 587.381,Z 194.884,A -85,B 0,C 180,E1 -1543.514,E2 -1543.514} C_VEL
LIN {X 0,Y 587.523,Z 175.171,A -85,B 0,C 180,E1 -1546.326,E2 -1546.326} C_VEL
LIN {X 0,Y 587.609,Z 157.787,A -85,B 0,C 180,E1 -1548.84,E2 -1548.84} C_VEL
LIN {X 0,Y 587.797,Z 139.161,A -85,B 0,C 180,E1 -1551.571,E2 -1551.571} C_VEL
LIN {X 0,Y 587.583,Z 134.14,A -85,B 0,C 180,E1 -1552.319,E2 -1552.319} C_VEL
LIN {X 0,Y 587.342,Z 132.823,A -85,B 0,C 180,E1 -1552.557,E2 -1552.557} C_VEL
LIN {X 0,Y 587.322,Z 132.825,A -85,B 0,C 180,E1 -1555.517,E2 -1555.517} C_VEL
LIN {X 0,Y 587.293,Z 132.824,A -85,B 0,C 180,E1 -1557.82,E2 -1557.82} C_VEL
LIN {X 0,Y 587.296,Z 132.823,A -85,B 0,C 180,E1 -1560.172,E2 -1560.172} C_VEL
LIN {X 0,Y 587.327,Z 132.824,A -85,B 0,C 180,E1 -1562.58,E2 -1562.58} C_VEL
LIN {X 0,Y 587.322,Z 132.827,A -85,B 0,C 180,E1 -1565.056,E2 -1565.056} C_VEL
LIN {X 0,Y 587.328,Z 132.819,A -85,B 0,C 180,E1 -1567.837,E2 -1567.837} C_VEL
LIN {X 0,Y 587.302,Z 132.825,A -85,B 0,C 180,E1 -1570.255,E2 -1570.255} C_VEL
LIN {X 0,Y 587.304,Z 132.826,A -85,B 0,C 180,E1 -1573.007,E2 -1573.007} C_VEL
LIN {X 0,Y 587.312,Z 132.824,A -85,B 0,C 180,E1 -1576.048,E2 -1576.048} C_VEL
LIN {X 0,Y 587.335,Z 132.821,A -85,B 0,C 180,E1 -1578.925,E2 -1578.925} C_VEL
LIN {X 0,Y 587.319,Z 132.82,A -85,B 0,C 180,E1 -1581.52,E2 -1581.52} C_VEL
LIN {X 0,Y 587.287,Z 132.831,A -85,B 0,C 180,E1 -1584.1,E2 -1584.1} C_VEL
LIN {X 0,Y 587.332,Z 132.823,A -85,B 0,C 180,E1 -1586.603,E2 -1586.603} C_VEL
LIN {X 0,Y 587.32,Z 132.821,A -85,B 0,C 180,E1 -1589.493,E2 -1589.493} C_VEL
LIN {X 0,Y 587.34,Z 132.824,A -85,B 0,C 180,E1 -1592.309,E2 -1592.309} C_VEL
LIN {X 0,Y 587.353,Z 132.818,A -85,B 0,C 180,E1 -1595.42,E2 -1595.42} C_VEL
LIN {X 0,Y 587.317,Z 132.825,A -85,B 0,C 180,E1 -1598.225,E2 -1598.225} C_VEL
LIN {X 0,Y 587.342,Z 132.819,A -85,B 0,C 180,E1 -1601.151,E2 -1601.151} C_VEL
LIN {X 0,Y 587.317,Z 132.825,A -85,B 0,C 180,E1 -1604.025,E2 -1604.025} C_VEL
LIN {X 0,Y 587.355,Z 132.818,A -85,B 0,C 180,E1 -1606.154,E2 -1606.154} C_VEL
LIN {X 0,Y 587.338,Z 132.82,A -85,B 0,C 180,E1 -1608.962,E2 -1608.962} C_VEL
LIN {X 0,Y 587.365,Z 132.82,A -85,B 0,C 180,E1 -1611.745,E2 -1611.745} C_VEL
LIN {X 0,Y 587.354,Z 132.816,A -85,B 0,C 180,E1 -1614.507,E2 -1614.507} C_VEL
LIN {X 0,Y 587.374,Z 132.823,A -85,B 0,C 180,E1 -1617.257,E2 -1617.257} C_VEL
LIN {X 0,Y 587.383,Z 132.813,A -85,B 0,C 180,E1 -1620,E2 -1620} C_VEL
LIN {X 0,Y 587.363,Z 132.819,A -85,B 0,C 180,E1 -1622.743,E2 -1622.743} C_VEL
LIN {X 0,Y 587.365,Z 132.818,A -85,B 0,C 180,E1 -1625.493,E2 -1625.493} C_VEL
LIN {X 0,Y 587.363,Z 132.816,A -85,B 0,C 180,E1 -1628.255,E2 -1628.255} C_VEL
LIN {X 0,Y 587.348,Z 132.823,A -85,B 0,C 180,E1 -1631.134,E2 -1631.134} C_VEL
LIN {X 0,Y 587.365,Z 132.817,A -85,B 0,C 180,E1 -1634.26,E2 -1634.26} C_VEL
LIN {X 0,Y 587.349,Z 132.818,A -85,B 0,C 180,E1 -1637.406,E2 -1637.406} C_VEL
LIN {X 0,Y 587.309,Z 132.824,A -85,B 0,C 180,E1 -1638.3,E2 -1638.3} C_VEL
LIN {X 0,Y 586.667,Z 132.909,A -85,B 0,C 180,E1 -1638.872,E2 -1638.872} C_VEL
LIN {X 0,Y 583.843,Z 133.259,A -85,B 0,C 180,E1 -1639.801,E2 -1639.801} C_VEL
LIN {X 0,Y 581.433,Z 133.563,A -85,B 0,C 180,E1 -1640.548,E2 -1640.548} C_VEL
LIN {X 0,Y 580.38,Z 133.687,A -85,B 0,C 180,E1 -1641.124,E2 -1641.124} C_VEL
LIN {X 0,Y 580.285,Z 133.697,A -85,B 0,C 180,E1 -1641.319,E2 -1641.319} C_VEL
LIN {X 0,Y 580.278,Z 133.697,A -85,B 0,C 180,E1 -1643.558,E2 -1643.558} C_VEL
LIN {X 0,Y 580.292,Z 133.697,A -85,B 0,C 180,E1 -1645.849,E2 -1645.849} C_VEL
LIN {X 0,Y 580.3,Z 133.701,A -85,B 0,C 180,E1 -1648.186,E2 -1648.186} C_VEL
LIN {X 0,Y 580.284,Z 133.701,A -85,B 0,C 180,E1 -1650.695,E2 -1650.695} C_VEL
LIN {X 0,Y 580.305,Z 133.694,A -85,B 0,C 180,E1 -1653.317,E2 -1653.317} C_VEL
LIN {X 0,Y 580.246,Z 133.705,A -85,B 0,C 180,E1 -1655.756,E2 -1655.756} C_VEL
LIN {X 0,Y 580.291,Z 133.705,A -85,B 0,C 180,E1 -1658.146,E2 -1658.146} C_VEL
LIN {X 0,Y 580.301,Z 133.695,A -85,B 0,C 180,E1 -1660.843,E2 -1660.843} C_VEL
LIN {X 0,Y 580.281,Z 133.703,A -85,B 0,C 180,E1 -1663.658,E2 -1663.658} C_VEL
LIN {X 0,Y 580.279,Z 133.698,A -85,B 0,C 180,E1 -1666.609,E2 -1666.609} C_VEL
LIN {X 0,Y 580.3,Z 133.696,A -85,B 0,C 180,E1 -1669.157,E2 -1669.157} C_VEL
LIN {X 0,Y 580.291,Z 133.702,A -85,B 0,C 180,E1 -1671.927,E2 -1671.927} C_VEL
LIN {X 0,Y 580.252,Z 133.701,A -85,B 0,C 180,E1 -1674.453,E2 -1674.453} C_VEL
LIN {X 0,Y 580.291,Z 133.698,A -85,B 0,C 180,E1 -1676.975,E2 -1676.975} C_VEL
LIN {X 0,Y 580.289,Z 133.706,A -85,B 0,C 180,E1 -1679.425,E2 -1679.425} C_VEL
LIN {X 0,Y 580.294,Z 133.696,A -85,B 0,C 180,E1 -1682.143,E2 -1682.143} C_VEL
LIN {X 0,Y 580.324,Z 133.702,A -85,B 0,C 180,E1 -1685.27,E2 -1685.27} C_VEL
LIN {X 0,Y 580.27,Z 133.7,A -85,B 0,C 180,E1 -1687.947,E2 -1687.947} C_VEL
LIN {X 0,Y 580.337,Z 133.813,A -85,B 0,C 180,E1 -1690.064,E2 -1690.064} C_VEL
LIN {X 0,Y 580.553,Z 140.901,A -85,B 0,C 180,E1 -1691.289,E2 -1691.289} C_VEL
LIN {X 0,Y 580.424,Z 157.954,A -85,B 0,C 180,E1 -1694.191,E2 -1694.191} C_VEL
LIN {X 0,Y 580.361,Z 171.232,A -85,B 0,C 180,E1 -1696.4,E2 -1696.4} C_VEL
LIN {X 0,Y 580.97,Z 177.263,A -85,B 0,C 180,E1 -1696.49,E2 -1696.49} C_VEL
LIN {X 0,Y 580.829,Z 277.912,A -85,B 0,C 180,E1 -1697.753,E2 -1697.753} C_VEL
LIN {X 0,Y 580.721,Z 291.188,A -85,B 0,C 180,E1 -1698.061,E2 -1698.061} C_VEL
LIN {X 0,Y 580.651,Z 303.352,A -85,B 0,C 180,E1 -1698.48,E2 -1698.48} C_VEL
LIN {X 0,Y 580.554,Z 314.791,A -85,B 0,C 180,E1 -1699.008,E2 -1699.008} C_VEL
LIN {X 0,Y 580.447,Z 326.542,A -85,B 0,C 180,E1 -1699.712,E2 -1699.712} C_VEL
LIN {X 0,Y 580.346,Z 337.058,A -85,B 0,C 180,E1 -1700.503,E2 -1700.503} C_VEL
LIN {X 0,Y 580.272,Z 345.658,A -85,B 0,C 180,E1 -1701.292,E2 -1701.292} C_VEL
LIN {X 0,Y 580.222,Z 353.581,A -85,B 0,C 180,E1 -1702.168,E2 -1702.168} C_VEL
LIN {X 0,Y 580.168,Z 361.285,A -85,B 0,C 180,E1 -1703.21,E2 -1703.21} C_VEL
LIN {X 0,Y 580.139,Z 368.446,A -85,B 0,C 180,E1 -1704.438,E2 -1704.438} C_VEL
LIN {X 0,Y 580.108,Z 373.188,A -85,B 0,C 180,E1 -1705.483,E2 -1705.483} C_VEL
LIN {X 0,Y 580.123,Z 376.822,A -85,B 0,C 180,E1 -1706.527,E2 -1706.527} C_VEL
LIN {X 0,Y 580.043,Z 378.699,A -85,B 0,C 180,E1 -1707.222,E2 -1707.222} C_VEL
LIN {X 0,Y 580.04,Z 380.127,A -85,B 0,C 180,E1 -1707.917,E2 -1707.917} C_VEL
LIN {X 0,Y 580.041,Z 381.755,A -85,B 0,C 180,E1 -1709.306,E2 -1709.306} C_VEL
LIN {X 0,Y 580.038,Z 381.996,A -85,B 0,C 180,E1 -1710,E2 -1710} C_VEL
LIN {X 0,Y 580.04,Z 381.815,A -85,B 0,C 180,E1 -1710.694,E2 -1710.694} C_VEL
LIN {X 0,Y 580.04,Z 380.271,A -85,B 0,C 180,E1 -1712.083,E2 -1712.083} C_VEL
LIN {X 0,Y 580.044,Z 378.91,A -85,B 0,C 180,E1 -1712.778,E2 -1712.778} C_VEL
LIN {X 0,Y 580.11,Z 376.034,A -85,B 0,C 180,E1 -1713.821,E2 -1713.821} C_VEL
LIN {X 0,Y 580.053,Z 372.134,A -85,B 0,C 180,E1 -1714.865,E2 -1714.865} C_VEL
LIN {X 0,Y 580.162,Z 367.102,A -85,B 0,C 180,E1 -1715.91,E2 -1715.91} C_VEL
LIN {X 0,Y 580.158,Z 360.78,A -85,B 0,C 180,E1 -1716.958,E2 -1716.958} C_VEL
LIN {X 0,Y 580.241,Z 352.86,A -85,B 0,C 180,E1 -1718.007,E2 -1718.007} C_VEL
LIN {X 0,Y 580.308,Z 343.011,A -85,B 0,C 180,E1 -1719.058,E2 -1719.058} C_VEL
LIN {X 0,Y 580.418,Z 332.694,A -85,B 0,C 180,E1 -1719.936,E2 -1719.936} C_VEL
LIN {X 0,Y 580.511,Z 321.055,A -85,B 0,C 180,E1 -1720.727,E2 -1720.727} C_VEL
LIN {X 0,Y 580.649,Z 309.084,A -85,B 0,C 180,E1 -1721.361,E2 -1721.361} C_VEL
LIN {X 0,Y 580.677,Z 296.199,A -85,B 0,C 180,E1 -1721.873,E2 -1721.873} C_VEL
LIN {X 0,Y 580.778,Z 283.552,A -85,B 0,C 180,E1 -1722.226,E2 -1722.226} C_VEL
LIN {X 0,Y 580.864,Z 270.367,A -85,B 0,C 180,E1 -1722.446,E2 -1722.446} C_VEL
LIN {X 0,Y 580.864,Z 174.43,A -85,B 0,C 180,E1 -1723.638,E2 -1723.638} C_VEL
LIN {X 0,Y 580.351,Z 171.016,A -85,B 0,C 180,E1 -1723.704,E2 -1723.704} C_VEL
LIN {X 0,Y 580.448,Z 153.155,A -85,B 0,C 180,E1 -1726.712,E2 -1726.712} C_VEL
LIN {X 0,Y 580.567,Z 137.249,A -85,B 0,C 180,E1 -1729.429,E2 -1729.429} C_VEL
LIN {X 0,Y 580.297,Z 133.701,A -85,B 0,C 180,E1 -1730.053,E2 -1730.053} C_VEL
LIN {X 0,Y 580.265,Z 133.707,A -85,B 0,C 180,E1 -1733.001,E2 -1733.001} C_VEL
LIN {X 0,Y 580.306,Z 133.7,A -85,B 0,C 180,E1 -1735.08,E2 -1735.08} C_VEL
LIN {X 0,Y 580.297,Z 133.698,A -85,B 0,C 180,E1 -1738.186,E2 -1738.186} C_VEL
LIN {X 0,Y 580.278,Z 133.706,A -85,B 0,C 180,E1 -1740.693,E2 -1740.693} C_VEL
LIN {X 0,Y 580.285,Z 133.697,A -85,B 0,C 180,E1 -1743.313,E2 -1743.313} C_VEL
LIN {X 0,Y 580.246,Z 133.702,A -85,B 0,C 180,E1 -1745.756,E2 -1745.756} C_VEL
LIN {X 0,Y 580.288,Z 133.702,A -85,B 0,C 180,E1 -1748.146,E2 -1748.146} C_VEL
LIN {X 0,Y 580.298,Z 133.697,A -85,B 0,C 180,E1 -1750.843,E2 -1750.843} C_VEL
LIN {X 0,Y 580.28,Z 133.699,A -85,B 0,C 180,E1 -1753.657,E2 -1753.657} C_VEL
LIN {X 0,Y 580.277,Z 133.7,A -85,B 0,C 180,E1 -1756.609,E2 -1756.609} C_VEL
LIN {X 0,Y 580.3,Z 133.695,A -85,B 0,C 180,E1 -1759.156,E2 -1759.156} C_VEL
LIN {X 0,Y 580.291,Z 133.705,A -85,B 0,C 180,E1 -1761.927,E2 -1761.927} C_VEL
LIN {X 0,Y 580.251,Z 133.703,A -85,B 0,C 180,E1 -1764.452,E2 -1764.452} C_VEL
LIN {X 0,Y 580.291,Z 133.696,A -85,B 0,C 180,E1 -1766.975,E2 -1766.975} C_VEL
LIN {X 0,Y 580.296,Z 133.7,A -85,B 0,C 180,E1 -1769.425,E2 -1769.425} C_VEL
LIN {X 0,Y 580.298,Z 133.698,A -85,B 0,C 180,E1 -1772.141,E2 -1772.141} C_VEL
LIN {X 0,Y 580.321,Z 133.697,A -85,B 0,C 180,E1 -1775.27,E2 -1775.27} C_VEL
LIN {X 0,Y 580.274,Z 133.701,A -85,B 0,C 180,E1 -1777.947,E2 -1777.947} C_VEL
LIN {X 0,Y 580.319,Z 133.695,A -85,B 0,C 180,E1 -1780.914,E2 -1780.914} C_VEL
LIN {X 0,Y 580.277,Z 133.7,A -85,B 0,C 180,E1 -1783.825,E2 -1783.825} C_VEL
LIN {X 0,Y 580.325,Z 133.692,A -85,B 0,C 180,E1 -1785.983,E2 -1785.983} C_VEL
LIN {X 0,Y 580.304,Z 133.699,A -85,B 0,C 180,E1 -1788.827,E2 -1788.827} C_VEL
LIN {X 0,Y 580.326,Z 133.693,A -85,B 0,C 180,E1 -1791.644,E2 -1791.644} C_VEL
LIN {X 0,Y 580.329,Z 133.693,A -85,B 0,C 180,E1 -1794.44,E2 -1794.44} C_VEL
LIN {X 0,Y 580.334,Z 133.695,A -85,B 0,C 180,E1 -1797.223,E2 -1797.223} C_VEL
LIN {X 0,Y 580.352,Z 133.689,A -85,B 0,C 180,E1 -1800,E2 -1800} C_VEL
LIN {X 0,Y 580.339,Z 133.699,A -85,B 0,C 180,E1 -1802.777,E2 -1802.777} C_VEL
LIN {X 0,Y 580.323,Z 133.692,A -85,B 0,C 180,E1 -1805.56,E2 -1805.56} C_VEL
LIN {X 0,Y 580.328,Z 133.698,A -85,B 0,C 180,E1 -1808.356,E2 -1808.356} C_VEL
LIN {X 0,Y 580.299,Z 133.696,A -85,B 0,C 180,E1 -1811.191,E2 -1811.191} C_VEL
LIN {X 0,Y 580.323,Z 133.696,A -85,B 0,C 180,E1 -1814.017,E2 -1814.017} C_VEL
LIN {X 0,Y 580.312,Z 133.695,A -85,B 0,C 180,E1 -1816.914,E2 -1816.914} C_VEL
LIN {X 0,Y 580.285,Z 133.701,A -85,B 0,C 180,E1 -1819.823,E2 -1819.823} C_VEL
LIN {X 0,Y 580.271,Z 133.707,A -85,B 0,C 180,E1 -1822.053,E2 -1822.053} C_VEL
LIN {X 0,Y 580.305,Z 133.694,A -85,B 0,C 180,E1 -1825.08,E2 -1825.08} C_VEL
LIN {X 0,Y 580.29,Z 133.702,A -85,B 0,C 180,E1 -1828.186,E2 -1828.186} C_VEL
LIN {X 0,Y 580.279,Z 133.698,A -85,B 0,C 180,E1 -1830.694,E2 -1830.694} C_VEL
LIN {X 0,Y 580.301,Z 133.697,A -85,B 0,C 180,E1 -1833.316,E2 -1833.316} C_VEL
LIN {X 0,Y 580.243,Z 133.712,A -85,B 0,C 180,E1 -1835.756,E2 -1835.756} C_VEL
LIN {X 0,Y 580.283,Z 133.699,A -85,B 0,C 180,E1 -1838.147,E2 -1838.147} C_VEL
LIN {X 0,Y 580.296,Z 133.696,A -85,B 0,C 180,E1 -1840.844,E2 -1840.844} C_VEL
LIN {X 0,Y 580.269,Z 133.706,A -85,B 0,C 180,E1 -1843.659,E2 -1843.659} C_VEL
LIN {X 0,Y 580.243,Z 133.702,A -85,B 0,C 180,E1 -1846.613,E2 -1846.613} C_VEL
LIN {X 0,Y 580.293,Z 133.703,A -85,B 0,C 180,E1 -1849.156,E2 -1849.156} C_VEL
LIN {X 0,Y 580.283,Z 133.698,A -85,B 0,C 180,E1 -1851.928,E2 -1851.928} C_VEL
LIN {X 0,Y 580.247,Z 133.702,A -85,B 0,C 180,E1 -1854.453,E2 -1854.453} C_VEL
LIN {X 0,Y 580.284,Z 133.705,A -85,B 0,C 180,E1 -1856.975,E2 -1856.975} C_VEL
LIN {X 0,Y 580.271,Z 133.703,A -85,B 0,C 180,E1 -1859.424,E2 -1859.424} C_VEL
LIN {X 0,Y 580.246,Z 133.702,A -85,B 0,C 180,E1 -1862.152,E2 -1862.152} C_VEL
LIN {X 0,Y 580.278,Z 133.707,A -85,B 0,C 180,E1 -1864.919,E2 -1864.919} C_VEL
LIN {X 0,Y 580.307,Z 133.819,A -85,B 0,C 180,E1 -1867.363,E2 -1867.363} C_VEL
LIN {X 0,Y 580.85,Z 139.013,A -85,B 0,C 180,E1 -1868.158,E2 -1868.158} C_VEL
LIN {X 0,Y 580.669,Z 157.787,A -85,B 0,C 180,E1 -1870.926,E2 -1870.926} C_VEL
LIN {X 0,Y 580.527,Z 176.414,A -85,B 0,C 180,E1 -1873.652,E2 -1873.652} C_VEL
LIN {X 0,Y 580.393,Z 195.149,A -85,B 0,C 180,E1 -1876.342,E2 -1876.342} C_VEL
LIN {X 0,Y 580.956,Z 200.515,A -85,B 0,C 180,E1 -1876.422,E2 -1876.422} C_VEL
LIN {X 0,Y 580.786,Z 302.95,A -85,B 0,C 180,E1 -1877.708,E2 -1877.708} C_VEL
LIN {X 0,Y 580.727,Z 316.221,A -85,B 0,C 180,E1 -1878.017,E2 -1878.017} C_VEL
LIN {X 0,Y 580.649,Z 328.377,A -85,B 0,C 180,E1 -1878.436,E2 -1878.436} C_VEL
LIN {X 0,Y 580.556,Z 340.629,A -85,B 0,C 180,E1 -1879.009,E2 -1879.009} C_VEL
LIN {X 0,Y 580.441,Z 352.202,A -85,B 0,C 180,E1 -1879.712,E2 -1879.712} C_VEL
LIN {X 0,Y 580.345,Z 362.602,A -85,B 0,C 180,E1 -1880.503,E2 -1880.503} C_VEL
LIN {X 0,Y 580.271,Z 371.113,A -85,B 0,C 180,E1 -1881.292,E2 -1881.292} C_VEL
LIN {X 0,Y 580.222,Z 378.961,A -85,B 0,C 180,E1 -1882.168,E2 -1882.168} C_VEL
LIN {X 0,Y 580.153,Z 386.651,A -85,B 0,C 180,E1 -1883.222,E2 -1883.222} C_VEL
LIN {X 0,Y 580.139,Z 393.68,A -85,B 0,C 180,E1 -1884.439,E2 -1884.439} C_VEL
LIN {X 0,Y 580.108,Z 398.372,A -85,B 0,C 180,E1 -1885.483,E2 -1885.483} C_VEL
LIN {X 0,Y 580.123,Z 401.957,A -85,B 0,C 180,E1 -1886.527,E2 -1886.527} C_VEL
LIN {X 0,Y 580.043,Z 403.808,A -85,B 0,C 180,E1 -1887.222,E2 -1887.222} C_VEL
LIN {X 0,Y 580.04,Z 405.198,A -85,B 0,C 180,E1 -1887.917,E2 -1887.917} C_VEL
LIN {X 0,Y 580.04,Z 406.785,A -85,B 0,C 180,E1 -1889.306,E2 -1889.306} C_VEL
LIN {X 0,Y 580.037,Z 407,A -85,B 0,C 180,E1 -1890,E2 -1890} C_VEL
LIN {X 0,Y 580.047,Z 406.186,A -85,B 0,C 180,E1 -1891.389,E2 -1891.389} C_VEL
LIN {X 0,Y 580.04,Z 405.199,A -85,B 0,C 180,E1 -1892.083,E2 -1892.083} C_VEL
LIN {X 0,Y 580.043,Z 403.81,A -85,B 0,C 180,E1 -1892.778,E2 -1892.778} C_VEL
LIN {X 0,Y 580.11,Z 400.896,A -85,B 0,C 180,E1 -1893.821,E2 -1893.821} C_VEL
LIN {X 0,Y 580.053,Z 396.949,A -85,B 0,C 180,E1 -1894.865,E2 -1894.865} C_VEL
LIN {X 0,Y 580.139,Z 390.877,A -85,B 0,C 180,E1 -1896.085,E2 -1896.085} C_VEL
LIN {X 0,Y 580.184,Z 384.237,A -85,B 0,C 180,E1 -1897.132,E2 -1897.132} C_VEL
LIN {X 0,Y 580.25,Z 375.991,A -85,B 0,C 180,E1 -1898.182,E2 -1898.182} C_VEL
LIN {X 0,Y 580.308,Z 367.539,A -85,B 0,C 180,E1 -1899.058,E2 -1899.058} C_VEL
LIN {X 0,Y 580.422,Z 357.098,A -85,B 0,C 180,E1 -1899.936,E2 -1899.936} C_VEL
LIN {X 0,Y 580.506,Z 346.754,A -85,B 0,C 180,E1 -1900.639,E2 -1900.639} C_VEL
LIN {X 0,Y 580.596,Z 335.246,A -85,B 0,C 180,E1 -1901.264,E2 -1901.264} C_VEL
LIN {X 0,Y 580.683,Z 322.472,A -85,B 0,C 180,E1 -1901.785,E2 -1901.785} C_VEL
LIN {X 0,Y 580.755,Z 309.434,A -85,B 0,C 180,E1 -1902.16,E2 -1902.16} C_VEL
LIN {X 0,Y 580.839,Z 297.085,A -85,B 0,C 180,E1 -1902.38,E2 -1902.38} C_VEL
LIN {X 0,Y 580.784,Z 197.727,A -85,B 0,C 180,E1 -1903.616,E2 -1903.616} C_VEL
LIN {X 0,Y 580.386,Z 194.884,A -85,B 0,C 180,E1 -1903.68,E2 -1903.68} C_VEL
LIN {X 0,Y 580.533,Z 173.93,A -85,B 0,C 180,E1 -1906.71,E2 -1906.71} C_VEL
LIN {X 0,Y 580.665,Z 156.568,A -85,B 0,C 180,E1 -1909.254,E2 -1909.254} C_VEL
LIN {X 0,Y 580.837,Z 137.757,A -85,B 0,C 180,E1 -1912.03,E2 -1912.03} C_VEL
LIN {X 0,Y 580.3,Z 133.701,A -85,B 0,C 180,E1 -1912.661,E2 -1912.661} C_VEL
LIN {X 0,Y 580.26,Z 133.702,A -85,B 0,C 180,E1 -1915.85,E2 -1915.85} C_VEL
LIN {X 0,Y 580.238,Z 133.702,A -85,B 0,C 180,E1 -1918.189,E2 -1918.189} C_VEL
LIN {X 0,Y 580.262,Z 133.704,A -85,B 0,C 180,E1 -1920.69,E2 -1920.69} C_VEL
LIN {X 0,Y 580.279,Z 133.701,A -85,B 0,C 180,E1 -1923.312,E2 -1923.312} C_VEL
LIN {X 0,Y 580.241,Z 133.702,A -85,B 0,C 180,E1 -1925.755,E2 -1925.755} C_VEL
LIN {X 0,Y 580.281,Z 133.698,A -85,B 0,C 180,E1 -1928.147,E2 -1928.147} C_VEL
LIN {X 0,Y 580.293,Z 133.703,A -85,B 0,C 180,E1 -1930.844,E2 -1930.844} C_VEL
LIN {X 0,Y 580.241,Z 133.702,A -85,B 0,C 180,E1 -1933.661,E2 -1933.661} C_VEL
LIN {X 0,Y 580.267,Z 133.708,A -85,B 0,C 180,E1 -1936.61,E2 -1936.61} C_VEL
LIN {X 0,Y 580.297,Z 133.696,A -85,B 0,C 180,E1 -1939.156,E2 -1939.156} C_VEL
LIN {X 0,Y 580.285,Z 133.7,A -85,B 0,C 180,E1 -1941.927,E2 -1941.927} C_VEL
LIN {X 0,Y 580.249,Z 133.708,A -85,B 0,C 180,E1 -1944.452,E2 -1944.452} C_VEL
LIN {X 0,Y 580.287,Z 133.697,A -85,B 0,C 180,E1 -1946.975,E2 -1946.975} C_VEL
LIN {X 0,Y 580.282,Z 133.698,A -85,B 0,C 180,E1 -1949.424,E2 -1949.424} C_VEL
LIN {X 0,Y 580.287,Z 133.705,A -85,B 0,C 180,E1 -1952.143,E2 -1952.143} C_VEL
LIN {X 0,Y 580.321,Z 133.693,A -85,B 0,C 180,E1 -1955.27,E2 -1955.27} C_VEL
LIN {X 0,Y 580.269,Z 133.708,A -85,B 0,C 180,E1 -1957.947,E2 -1957.947} C_VEL
LIN {X 0,Y 580.292,Z 133.696,A -85,B 0,C 180,E1 -1960.913,E2 -1960.913} C_VEL
LIN {X 0,Y 580.268,Z 133.707,A -85,B 0,C 180,E1 -1963.825,E2 -1963.825} C_VEL
LIN {X 0,Y 580.324,Z 133.696,A -85,B 0,C 180,E1 -1965.983,E2 -1965.983} C_VEL
LIN {X 0,Y 580.305,Z 133.695,A -85,B 0,C 180,E1 -1968.827,E2 -1968.827} C_VEL
LIN {X 0,Y 580.328,Z 133.698,A -85,B 0,C 180,E1 -1971.644,E2 -1971.644} C_VEL
LIN {X 0,Y 580.322,Z 133.692,A -85,B 0,C 180,E1 -1974.44,E2 -1974.44} C_VEL
LIN {X 0,Y 580.346,Z 133.69,A -85,B 0,C 180,E1 -1977.918,E2 -1977.918} C_VEL
LIN {X 0,Y 580.353,Z 133.69,A -85,B 0,C 180,E1 -1980.694,E2 -1980.694} C_VEL
LIN {X 0,Y 580.288,Z 133.701,A -85,B 0,C 180,E1 -1983.472,E2 -1983.472} C_VEL
LIN {X 0,Y 580.331,Z 133.693,A -85,B 0,C 180,E1 -1985.56,E2 -1985.56} C_VEL
LIN {X 0,Y 580.326,Z 133.693,A -85,B 0,C 180,E1 -1988.356,E2 -1988.356} C_VEL
LIN {X 0,Y 580.3,Z 133.7,A -85,B 0,C 180,E1 -1991.191,E2 -1991.191} C_VEL
LIN {X 0,Y 580.326,Z 133.692,A -85,B 0,C 180,E1 -1994.017,E2 -1994.017} C_VEL
LIN {X 0,Y 580.312,Z 133.7,A -85,B 0,C 180,E1 -1996.914,E2 -1996.914} C_VEL
LIN {X 0,Y 580.304,Z 133.695,A -85,B 0,C 180,E1 -1999.822,E2 -1999.822} C_VEL
LIN {X 0,Y 580.285,Z 133.697,A -85,B 0,C 180,E1 -2001.319,E2 -2001.319} C_VEL
LIN {X 0,Y 579.587,Z 133.785,A -85,B 0,C 180,E1 -2001.899,E2 -2001.899} C_VEL
LIN {X 0,Y 576.71,Z 134.147,A -85,B 0,C 180,E1 -2002.838,E2 -2002.838} C_VEL
LIN {X 0,Y 574.315,Z 134.443,A -85,B 0,C 180,E1 -2003.595,E2 -2003.595} C_VEL
LIN {X 0,Y 573.316,Z 134.569,A -85,B 0,C 180,E1 -2004.179,E2 -2004.179} C_VEL
LIN {X 0,Y 573.249,Z 134.577,A -85,B 0,C 180,E1 -2004.376,E2 -2004.376} C_VEL
LIN {X 0,Y 573.251,Z 134.575,A -85,B 0,C 180,E1 -2006.976,E2 -2006.976} C_VEL
LIN {X 0,Y 573.247,Z 134.573,A -85,B 0,C 180,E1 -2009.488,E2 -2009.488} C_VEL
LIN {X 0,Y 573.255,Z 134.576,A -85,B 0,C 180,E1 -2012.645,E2 -2012.645} C_VEL
LIN {X 0,Y 573.207,Z 134.578,A -85,B 0,C 180,E1 -2015.188,E2 -2015.188} C_VEL
LIN {X 0,Y 573.238,Z 134.58,A -85,B 0,C 180,E1 -2017.808,E2 -2017.808} C_VEL
LIN {X 0,Y 573.271,Z 134.573,A -85,B 0,C 180,E1 -2020.528,E2 -2020.528} C_VEL
LIN {X 0,Y 573.246,Z 134.579,A -85,B 0,C 180,E1 -2023.669,E2 -2023.669} C_VEL
LIN {X 0,Y 573.242,Z 134.574,A -85,B 0,C 180,E1 -2026.641,E2 -2026.641} C_VEL
LIN {X 0,Y 573.246,Z 134.579,A -85,B 0,C 180,E1 -2029.475,E2 -2029.475} C_VEL
LIN {X 0,Y 573.237,Z 134.577,A -85,B 0,C 180,E1 -2032.193,E2 -2032.193} C_VEL
LIN {X 0,Y 573.235,Z 134.579,A -85,B 0,C 180,E1 -2035.229,E2 -2035.229} C_VEL
LIN {X 0,Y 573.242,Z 134.575,A -85,B 0,C 180,E1 -2038.185,E2 -2038.185} C_VEL
LIN {X 0,Y 573.262,Z 134.572,A -85,B 0,C 180,E1 -2040.634,E2 -2040.634} C_VEL
LIN {X 0,Y 573.238,Z 134.582,A -85,B 0,C 180,E1 -2043.508,E2 -2043.508} C_VEL
LIN {X 0,Y 573.225,Z 134.577,A -85,B 0,C 180,E1 -2046.134,E2 -2046.134} C_VEL
LIN {X 0,Y 573.256,Z 134.582,A -85,B 0,C 180,E1 -2049.174,E2 -2049.174} C_VEL
LIN {X 0,Y 573.287,Z 134.697,A -85,B 0,C 180,E1 -2049.971,E2 -2049.971} C_VEL
LIN {X 0,Y 573.576,Z 140.877,A -85,B 0,C 180,E1 -2051.052,E2 -2051.052} C_VEL
LIN {X 0,Y 573.411,Z 156.892,A -85,B 0,C 180,E1 -2053.809,E2 -2053.809} C_VEL
LIN {X 0,Y 573.318,Z 171.279,A -85,B 0,C 180,E1 -2056.229,E2 -2056.229} C_VEL
LIN {X 0,Y 574.082,Z 177.308,A -85,B 0,C 180,E1 -2056.324,E2 -2056.324} C_VEL
LIN {X 0,Y 573.9,Z 277.94,A -85,B 0,C 180,E1 -2057.603,E2 -2057.603} C_VEL
LIN {X 0,Y 573.781,Z 291.206,A -85,B 0,C 180,E1 -2057.914,E2 -2057.914} C_VEL
LIN {X 0,Y 573.708,Z 303.367,A -85,B 0,C 180,E1 -2058.339,E2 -2058.339} C_VEL
LIN {X 0,Y 573.583,Z 314.902,A -85,B 0,C 180,E1 -2058.878,E2 -2058.878} C_VEL
LIN {X 0,Y 573.433,Z 326.548,A -85,B 0,C 180,E1 -2059.585,E2 -2059.585} C_VEL
LIN {X 0,Y 573.334,Z 337.067,A -85,B 0,C 180,E1 -2060.386,E2 -2060.386} C_VEL
LIN {X 0,Y 573.241,Z 345.664,A -85,B 0,C 180,E1 -2061.185,E2 -2061.185} C_VEL
LIN {X 0,Y 573.161,Z 353.586,A -85,B 0,C 180,E1 -2062.071,E2 -2062.071} C_VEL
LIN {X 0,Y 573.093,Z 361.524,A -85,B 0,C 180,E1 -2063.163,E2 -2063.163} C_VEL
LIN {X 0,Y 573.071,Z 368.449,A -85,B 0,C 180,E1 -2064.37,E2 -2064.37} C_VEL
LIN {X 0,Y 573.028,Z 373.19,A -85,B 0,C 180,E1 -2065.427,E2 -2065.427} C_VEL
LIN {X 0,Y 573.022,Z 376.824,A -85,B 0,C 180,E1 -2066.484,E2 -2066.484} C_VEL
LIN {X 0,Y 572.959,Z 378.701,A -85,B 0,C 180,E1 -2067.188,E2 -2067.188} C_VEL
LIN {X 0,Y 572.94,Z 380.127,A -85,B 0,C 180,E1 -2067.891,E2 -2067.891} C_VEL
LIN {X 0,Y 572.941,Z 381.756,A -85,B 0,C 180,E1 -2069.297,E2 -2069.297} C_VEL
LIN {X 0,Y 572.939,Z 381.996,A -85,B 0,C 180,E1 -2070,E2 -2070} C_VEL
LIN {X 0,Y 572.94,Z 381.815,A -85,B 0,C 180,E1 -2070.703,E2 -2070.703} C_VEL
LIN {X 0,Y 572.94,Z 380.269,A -85,B 0,C 180,E1 -2072.109,E2 -2072.109} C_VEL
LIN {X 0,Y 572.96,Z 378.908,A -85,B 0,C 180,E1 -2072.812,E2 -2072.812} C_VEL
LIN {X 0,Y 573.015,Z 376.031,A -85,B 0,C 180,E1 -2073.868,E2 -2073.868} C_VEL
LIN {X 0,Y 572.963,Z 372.132,A -85,B 0,C 180,E1 -2074.926,E2 -2074.926} C_VEL
LIN {X 0,Y 573.076,Z 367.1,A -85,B 0,C 180,E1 -2075.983,E2 -2075.983} C_VEL
LIN {X 0,Y 573.083,Z 360.776,A -85,B 0,C 180,E1 -2077.044,E2 -2077.044} C_VEL
LIN {X 0,Y 573.175,Z 352.855,A -85,B 0,C 180,E1 -2078.106,E2 -2078.106} C_VEL
LIN {X 0,Y 573.287,Z 343.005,A -85,B 0,C 180,E1 -2079.17,E2 -2079.17} C_VEL
LIN {X 0,Y 573.421,Z 332.689,A -85,B 0,C 180,E1 -2080.058,E2 -2080.058} C_VEL
LIN {X 0,Y 573.509,Z 321.043,A -85,B 0,C 180,E1 -2080.86,E2 -2080.86} C_VEL
LIN {X 0,Y 573.658,Z 310.2,A -85,B 0,C 180,E1 -2081.449,E2 -2081.449} C_VEL
LIN {X 0,Y 573.733,Z 297.613,A -85,B 0,C 180,E1 -2081.97,E2 -2081.97} C_VEL
LIN {X 0,Y 573.861,Z 284.444,A -85,B 0,C 180,E1 -2082.353,E2 -2082.353} C_VEL
LIN {X 0,Y 573.944,Z 272.095,A -85,B 0,C 180,E1 -2082.576,E2 -2082.576} C_VEL
LIN {X 0,Y 574.038,Z 175.502,A -85,B 0,C 180,E1 -2083.79,E2 -2083.79} C_VEL
LIN {X 0,Y 573.31,Z 171.012,A -85,B 0,C 180,E1 -2083.875,E2 -2083.875} C_VEL
LIN {X 0,Y 573.453,Z 154.347,A -85,B 0,C 180,E1 -2086.716,E2 -2086.716} C_VEL
LIN {X 0,Y 573.551,Z 139.063,A -85,B 0,C 180,E1 -2089.348,E2 -2089.348} C_VEL
LIN {X 0,Y 573.285,Z 134.575,A -85,B 0,C 180,E1 -2090.169,E2 -2090.169} C_VEL
LIN {X 0,Y 573.215,Z 134.583,A -85,B 0,C 180,E1 -2093.139,E2 -2093.139} C_VEL
LIN {X 0,Y 573.25,Z 134.575,A -85,B 0,C 180,E1 -2095.41,E2 -2095.41} C_VEL
LIN {X 0,Y 573.248,Z 134.574,A -85,B 0,C 180,E1 -2098.028,E2 -2098.028} C_VEL
LIN {X 0,Y 573.24,Z 134.577,A -85,B 0,C 180,E1 -2100.176,E2 -2100.176} C_VEL
LIN {X 0,Y 573.254,Z 134.581,A -85,B 0,C 180,E1 -2102.645,E2 -2102.645} C_VEL
LIN {X 0,Y 573.207,Z 134.579,A -85,B 0,C 180,E1 -2105.188,E2 -2105.188} C_VEL
LIN {X 0,Y 573.236,Z 134.576,A -85,B 0,C 180,E1 -2107.807,E2 -2107.807} C_VEL
LIN {X 0,Y 573.246,Z 134.58,A -85,B 0,C 180,E1 -2110.525,E2 -2110.525} C_VEL
LIN {X 0,Y 573.241,Z 134.574,A -85,B 0,C 180,E1 -2113.359,E2 -2113.359} C_VEL
LIN {X 0,Y 573.245,Z 134.58,A -85,B 0,C 180,E1 -2116.331,E2 -2116.331} C_VEL
LIN {X 0,Y 573.26,Z 134.574,A -85,B 0,C 180,E1 -2119.476,E2 -2119.476} C_VEL
LIN {X 0,Y 573.237,Z 134.581,A -85,B 0,C 180,E1 -2122.192,E2 -2122.192} C_VEL
LIN {X 0,Y 573.235,Z 134.576,A -85,B 0,C 180,E1 -2125.228,E2 -2125.228} C_VEL
LIN {X 0,Y 573.251,Z 134.583,A -85,B 0,C 180,E1 -2127.772,E2 -2127.772} C_VEL
LIN {X 0,Y 573.264,Z 134.571,A -85,B 0,C 180,E1 -2130.634,E2 -2130.634} C_VEL
LIN {X 0,Y 573.251,Z 134.574,A -85,B 0,C 180,E1 -2133.024,E2 -2133.024} C_VEL
LIN {X 0,Y 573.275,Z 134.576,A -85,B 0,C 180,E1 -2135.366,E2 -2135.366} C_VEL
LIN {X 0,Y 573.229,Z 134.576,A -85,B 0,C 180,E1 -2138.419,E2 -2138.419} C_VEL
LIN {X 0,Y 573.278,Z 134.571,A -85,B 0,C 180,E1 -2140.728,E2 -2140.728} C_VEL
LIN {X 0,Y 573.249,Z 134.578,A -85,B 0,C 180,E1 -2143.622,E2 -2143.622} C_VEL
LIN {X 0,Y 573.272,Z 134.572,A -85,B 0,C 180,E1 -2145.807,E2 -2145.807} C_VEL
LIN {X 0,Y 573.262,Z 134.575,A -85,B 0,C 180,E1 -2148.745,E2 -2148.745} C_VEL
LIN {X 0,Y 573.282,Z 134.572,A -85,B 0,C 180,E1 -2151.54,E2 -2151.54} C_VEL
LIN {X 0,Y 573.297,Z 134.569,A -85,B 0,C 180,E1 -2154.372,E2 -2154.372} C_VEL
LIN {X 0,Y 573.314,Z 134.565,A -85,B 0,C 180,E1 -2157.892,E2 -2157.892} C_VEL
LIN {X 0,Y 573.335,Z 134.571,A -85,B 0,C 180,E1 -2160.702,E2 -2160.702} C_VEL
LIN {X 0,Y 573.305,Z 134.575,A -85,B 0,C 180,E1 -2162.811,E2 -2162.811} C_VEL
LIN {X 0,Y 573.292,Z 134.568,A -85,B 0,C 180,E1 -2165.628,E2 -2165.628} C_VEL
LIN {X 0,Y 573.284,Z 134.577,A -85,B 0,C 180,E1 -2168.46,E2 -2168.46} C_VEL
LIN {X 0,Y 573.271,Z 134.571,A -85,B 0,C 180,E1 -2171.312,E2 -2171.312} C_VEL
LIN {X 0,Y 573.281,Z 134.578,A -85,B 0,C 180,E1 -2174.424,E2 -2174.424} C_VEL
LIN {X 0,Y 573.257,Z 134.572,A -85,B 0,C 180,E1 -2177.112,E2 -2177.112} C_VEL
LIN {X 0,Y 573.239,Z 134.582,A -85,B 0,C 180,E1 -2180.077,E2 -2180.077} C_VEL
LIN {X 0,Y 573.234,Z 134.581,A -85,B 0,C 180,E1 -2182.338,E2 -2182.338} C_VEL
LIN {X 0,Y 573.247,Z 134.575,A -85,B 0,C 180,E1 -2185.41,E2 -2185.41} C_VEL
LIN {X 0,Y 573.229,Z 134.577,A -85,B 0,C 180,E1 -2188.565,E2 -2188.565} C_VEL
LIN {X 0,Y 573.221,Z 134.577,A -85,B 0,C 180,E1 -2190.994,E2 -2190.994} C_VEL
LIN {X 0,Y 573.262,Z 134.577,A -85,B 0,C 180,E1 -2193.524,E2 -2193.524} C_VEL
LIN {X 0,Y 573.192,Z 134.585,A -85,B 0,C 180,E1 -2196.053,E2 -2196.053} C_VEL
LIN {X 0,Y 573.241,Z 134.574,A -85,B 0,C 180,E1 -2198.702,E2 -2198.702} C_VEL
LIN {X 0,Y 573.223,Z 134.586,A -85,B 0,C 180,E1 -2201.592,E2 -2201.592} C_VEL
LIN {X 0,Y 573.222,Z 134.577,A -85,B 0,C 180,E1 -2204.335,E2 -2204.335} C_VEL
LIN {X 0,Y 573.236,Z 134.585,A -85,B 0,C 180,E1 -2207.359,E2 -2207.359} C_VEL
LIN {X 0,Y 573.233,Z 134.575,A -85,B 0,C 180,E1 -2210.392,E2 -2210.392} C_VEL
LIN {X 0,Y 573.251,Z 134.581,A -85,B 0,C 180,E1 -2213.078,E2 -2213.078} C_VEL
LIN {X 0,Y 573.251,Z 134.575,A -85,B 0,C 180,E1 -2215.67,E2 -2215.67} C_VEL
LIN {X 0,Y 573.225,Z 134.576,A -85,B 0,C 180,E1 -2218.184,E2 -2218.184} C_VEL
LIN {X 0,Y 573.233,Z 134.581,A -85,B 0,C 180,E1 -2220.633,E2 -2220.633} C_VEL
LIN {X 0,Y 573.214,Z 134.58,A -85,B 0,C 180,E1 -2223.513,E2 -2223.513} C_VEL
LIN {X 0,Y 573.197,Z 134.583,A -85,B 0,C 180,E1 -2226.133,E2 -2226.133} C_VEL
LIN {X 0,Y 573.279,Z 134.761,A -85,B 0,C 180,E1 -2227.236,E2 -2227.236} C_VEL
LIN {X 0,Y 573.894,Z 140.113,A -85,B 0,C 180,E1 -2228.068,E2 -2228.068} C_VEL
LIN {X 0,Y 573.704,Z 157.686,A -85,B 0,C 180,E1 -2230.685,E2 -2230.685} C_VEL
LIN {X 0,Y 573.533,Z 175.271,A -85,B 0,C 180,E1 -2233.279,E2 -2233.279} C_VEL
LIN {X 0,Y 573.399,Z 195.149,A -85,B 0,C 180,E1 -2236.172,E2 -2236.172} C_VEL
LIN {X 0,Y 574.052,Z 200.515,A -85,B 0,C 180,E1 -2236.256,E2 -2236.256} C_VEL
LIN {X 0,Y 573.859,Z 302.95,A -85,B 0,C 180,E1 -2237.557,E2 -2237.557} C_VEL
LIN {X 0,Y 573.778,Z 316.221,A -85,B 0,C 180,E1 -2237.869,E2 -2237.869} C_VEL
LIN {X 0,Y 573.679,Z 328.379,A -85,B 0,C 180,E1 -2238.294,E2 -2238.294} C_VEL
LIN {X 0,Y 573.56,Z 340.74,A -85,B 0,C 180,E1 -2238.879,E2 -2238.879} C_VEL
LIN {X 0,Y 573.428,Z 352.199,A -85,B 0,C 180,E1 -2239.585,E2 -2239.585} C_VEL
LIN {X 0,Y 573.332,Z 362.603,A -85,B 0,C 180,E1 -2240.386,E2 -2240.386} C_VEL
LIN {X 0,Y 573.241,Z 371.113,A -85,B 0,C 180,E1 -2241.185,E2 -2241.185} C_VEL
LIN {X 0,Y 573.161,Z 378.961,A -85,B 0,C 180,E1 -2242.071,E2 -2242.071} C_VEL
LIN {X 0,Y 573.072,Z 386.955,A -85,B 0,C 180,E1 -2243.185,E2 -2243.185} C_VEL
LIN {X 0,Y 573.07,Z 393.68,A -85,B 0,C 180,E1 -2244.37,E2 -2244.37} C_VEL
LIN {X 0,Y 573.028,Z 398.372,A -85,B 0,C 180,E1 -2245.428,E2 -2245.428} C_VEL
LIN {X 0,Y 573.022,Z 401.958,A -85,B 0,C 180,E1 -2246.484,E2 -2246.484} C_VEL
LIN {X 0,Y 572.959,Z 403.808,A -85,B 0,C 180,E1 -2247.188,E2 -2247.188} C_VEL
LIN {X 0,Y 572.946,Z 406.185,A -85,B 0,C 180,E1 -2248.594,E2 -2248.594} C_VEL
LIN {X 0,Y 572.938,Z 407,A -85,B 0,C 180,E1 -2250,E2 -2250} C_VEL
LIN {X 0,Y 572.946,Z 406.186,A -85,B 0,C 180,E1 -2251.406,E2 -2251.406} C_VEL
LIN {X 0,Y 572.94,Z 405.199,A -85,B 0,C 180,E1 -2252.109,E2 -2252.109} C_VEL
LIN {X 0,Y 572.959,Z 403.81,A -85,B 0,C 180,E1 -2252.812,E2 -2252.812} C_VEL
LIN {X 0,Y 573.015,Z 400.896,A -85,B 0,C 180,E1 -2253.868,E2 -2253.868} C_VEL
LIN {X 0,Y 572.963,Z 396.949,A -85,B 0,C 180,E1 -2254.926,E2 -2254.926} C_VEL
LIN {X 0,Y 573.065,Z 390.876,A -85,B 0,C 180,E1 -2256.16,E2 -2256.16} C_VEL
LIN {X 0,Y 573.119,Z 384.237,A -85,B 0,C 180,E1 -2257.221,E2 -2257.221} C_VEL
LIN {X 0,Y 573.201,Z 375.991,A -85,B 0,C 180,E1 -2258.283,E2 -2258.283} C_VEL
LIN {X 0,Y 573.287,Z 367.539,A -85,B 0,C 180,E1 -2259.17,E2 -2259.17} C_VEL
LIN {X 0,Y 573.427,Z 357.096,A -85,B 0,C 180,E1 -2260.058,E2 -2260.058} C_VEL
LIN {X 0,Y 573.543,Z 345.431,A -85,B 0,C 180,E1 -2260.853,E2 -2260.853} C_VEL
LIN {X 0,Y 573.651,Z 334.307,A -85,B 0,C 180,E1 -2261.446,E2 -2261.446} C_VEL
LIN {X 0,Y 573.758,Z 321.169,A -85,B 0,C 180,E1 -2261.974,E2 -2261.974} C_VEL
LIN {X 0,Y 573.833,Z 308.518,A -85,B 0,C 180,E1 -2262.331,E2 -2262.331} C_VEL
LIN {X 0,Y 573.937,Z 295.311,A -85,B 0,C 180,E1 -2262.554,E2 -2262.554} C_VEL
LIN {X 0,Y 573.912,Z 198.721,A -85,B 0,C 180,E1 -2263.77,E2 -2263.77} C_VEL
